LIN {X 0,Y 297.727,Z 299.631,A -85,B 0,C 180,E1 -16461.174,E2 -16461.174} C_VEL
LIN {X 0,Y 297.211,Z 303.349,A -85,B 0,C 180,E1 -16463.293,E2 -16463.293} C_VEL
LIN {X 0,Y 297,Z 305.074,A -85,B 0,C 180,E1 -16464.569,E2 -16464.569} C_VEL
LIN {X 0,Y 296.826,Z 306.468,A -85,B 0,C 180,E1 -16465.927,E2 -16465.927} C_VEL
LIN {X 0,Y 296.548,Z 308.073,A -85,B 0,C 180,E1 -16468.642,E2 -16468.642} C_VEL
LIN {X 0,Y 296.529,Z 308.304,A -85,B 0,C 180,E1 -16470,E2 -16470} C_VEL
LIN {X 0,Y 296.548,Z 308.111,A -85,B 0,C 180,E1 -16471.358,E2 -16471.358} C_VEL
LIN {X 0,Y 296.821,Z 306.556,A -85,B 0,C 180,E1 -16474.074,E2 -16474.074} C_VEL
LIN {X 0,Y 296.965,Z 305.201,A -85,B 0,C 180,E1 -16475.432,E2 -16475.432} C_VEL
LIN {X 0,Y 297.36,Z 302.335,A -85,B 0,C 180,E1 -16477.469,E2 -16477.469} C_VEL
LIN {X 0,Y 297.904,Z 298.45,A -85,B 0,C 180,E1 -16479.506,E2 -16479.506} C_VEL
LIN {X 0,Y 298.767,Z 293.434,A -85,B 0,C 180,E1 -16481.534,E2 -16481.534} C_VEL
LIN {X 0,Y 299.934,Z 287.114,A -85,B 0,C 180,E1 -16483.552,E2 -16483.552} C_VEL
LIN {X 0,Y 301.351,Z 279.205,A -85,B 0,C 180,E1 -16485.557,E2 -16485.557} C_VEL
LIN {X 0,Y 302.82,Z 271.138,A -85,B 0,C 180,E1 -16487.212,E2 -16487.212} C_VEL
LIN {X 0,Y 304.186,Z 261.302,A -85,B 0,C 180,E1 -16488.873,E2 -16488.873} C_VEL
LIN {X 0,Y 305.736,Z 250.222,A -85,B 0,C 180,E1 -16490.346,E2 -16490.346} C_VEL
LIN {X 0,Y 306.69,Z 242.741,A -85,B 0,C 180,E1 -16491.157,E2 -16491.157} C_VEL
LIN {X 0,Y 305.142,Z 232.366,A -85,B 0,C 180,E1 -16492.291,E2 -16492.291} C_VEL
LIN {X 0,Y 302.504,Z 220.449,A -85,B 0,C 180,E1 -16493.406,E2 -16493.406} C_VEL
LIN {X 0,Y 298.984,Z 208.375,A -85,B 0,C 180,E1 -16494.349,E2 -16494.349} C_VEL
LIN {X 0,Y 297.712,Z 203.982,A -85,B 0,C 180,E1 -16494.644,E2 -16494.644} C_VEL
LIN {X 0,Y 297.998,Z 200.351,A -85,B 0,C 180,E1 -16498.144,E2 -16498.144} C_VEL
LIN {X 0,Y 298.334,Z 196.579,A -85,B 0,C 180,E1 -16501.997,E2 -16501.997} C_VEL
LIN {X 0,Y 298.503,Z 194.178,A -85,B 0,C 180,E1 -16504.508,E2 -16504.508} C_VEL
LIN {X 0,Y 298.467,Z 191.246,A -85,B 0,C 180,E1 -16507.751,E2 -16507.751} C_VEL
LIN {X 0,Y 298.356,Z 190.321,A -85,B 0,C 180,E1 -16508.982,E2 -16508.982} C_VEL
LIN {X 0,Y 298.372,Z 190.319,A -85,B 0,C 180,E1 -16513.097,E2 -16513.097} C_VEL
LIN {X 0,Y 298.404,Z 190.316,A -85,B 0,C 180,E1 -16516.921,E2 -16516.921} C_VEL
LIN {X 0,Y 298.397,Z 190.317,A -85,B 0,C 180,E1 -16521.008,E2 -16521.008} C_VEL
LIN {X 0,Y 298.406,Z 190.313,A -85,B 0,C 180,E1 -16523.928,E2 -16523.928} C_VEL
LIN {X 0,Y 298.396,Z 190.313,A -85,B 0,C 180,E1 -16527.2,E2 -16527.2} C_VEL
LIN {X 0,Y 298.428,Z 190.312,A -85,B 0,C 180,E1 -16530.616,E2 -16530.616} C_VEL
LIN {X 0,Y 298.48,Z 190.302,A -85,B 0,C 180,E1 -16533.476,E2 -16533.476} C_VEL
LIN {X 0,Y 298.437,Z 190.309,A -85,B 0,C 180,E1 -16536.697,E2 -16536.697} C_VEL
LIN {X 0,Y 298.541,Z 190.295,A -85,B 0,C 180,E1 -16540.757,E2 -16540.757} C_VEL
LIN {X 0,Y 298.595,Z 190.289,A -85,B 0,C 180,E1 -16544.995,E2 -16544.995} C_VEL
LIN {X 0,Y 298.584,Z 190.291,A -85,B 0,C 180,E1 -16549.146,E2 -16549.146} C_VEL
LIN {X 0,Y 298.706,Z 190.276,A -85,B 0,C 180,E1 -16551.229,E2 -16551.229} C_VEL
LIN {X 0,Y 297.983,Z 190.365,A -85,B 0,C 180,E1 -16552.353,E2 -16552.353} C_VEL
LIN {X 0,Y 295.038,Z 190.732,A -85,B 0,C 180,E1 -16554.182,E2 -16554.182} C_VEL
LIN {X 0,Y 292.659,Z 191.031,A -85,B 0,C 180,E1 -16555.668,E2 -16555.668} C_VEL
LIN {X 0,Y 291.776,Z 191.14,A -85,B 0,C 180,E1 -16556.819,E2 -16556.819} C_VEL
LIN {X 0,Y 291.777,Z 191.142,A -85,B 0,C 180,E1 -16557.208,E2 -16557.208} C_VEL
LIN {X 0,Y 291.968,Z 191.114,A -85,B 0,C 180,E1 -16560,E2 -16560} C_VEL
LIN {X 0,Y 291.786,Z 191.139,A -85,B 0,C 180,E1 -16562.761,E2 -16562.761} C_VEL
LIN {X 0,Y 291.688,Z 191.154,A -85,B 0,C 180,E1 -16566.919,E2 -16566.919} C_VEL
LIN {X 0,Y 291.574,Z 191.164,A -85,B 0,C 180,E1 -16569.714,E2 -16569.714} C_VEL
LIN {X 0,Y 291.524,Z 191.171,A -85,B 0,C 180,E1 -16573.95,E2 -16573.95} C_VEL
LIN {X 0,Y 291.488,Z 191.177,A -85,B 0,C 180,E1 -16576.818,E2 -16576.818} C_VEL
LIN {X 0,Y 291.452,Z 191.181,A -85,B 0,C 180,E1 -16579.875,E2 -16579.875} C_VEL
LIN {X 0,Y 291.384,Z 191.191,A -85,B 0,C 180,E1 -16584.207,E2 -16584.207} C_VEL
LIN {X 0,Y 291.422,Z 191.183,A -85,B 0,C 180,E1 -16587.272,E2 -16587.272} C_VEL
LIN {X 0,Y 291.335,Z 191.196,A -85,B 0,C 180,E1 -16590.437,E2 -16590.437} C_VEL
LIN {X 0,Y 291.345,Z 191.197,A -85,B 0,C 180,E1 -16593.698,E2 -16593.698} C_VEL
LIN {X 0,Y 291.36,Z 191.194,A -85,B 0,C 180,E1 -16597.25,E2 -16597.25} C_VEL
LIN {X 0,Y 291.333,Z 191.197,A -85,B 0,C 180,E1 -16600.643,E2 -16600.643} C_VEL
LIN {X 0,Y 291.398,Z 191.4,A -85,B 0,C 180,E1 -16602.478,E2 -16602.478} C_VEL
LIN {X 0,Y 292.043,Z 195.349,A -85,B 0,C 180,E1 -16606.216,E2 -16606.216} C_VEL
LIN {X 0,Y 292.729,Z 199.137,A -85,B 0,C 180,E1 -16609.591,E2 -16609.591} C_VEL
LIN {X 0,Y 293.088,Z 202.423,A -85,B 0,C 180,E1 -16612.309,E2 -16612.309} C_VEL
LIN {X 0,Y 293.108,Z 205.65,A -85,B 0,C 180,E1 -16614.868,E2 -16614.868} C_VEL
LIN {X 0,Y 292.471,Z 209.913,A -85,B 0,C 180,E1 -16618.085,E2 -16618.085} C_VEL
LIN {X 0,Y 291.733,Z 215.231,A -85,B 0,C 180,E1 -16621.981,E2 -16621.981} C_VEL
LIN {X 0,Y 291.179,Z 219.113,A -85,B 0,C 180,E1 -16624.786,E2 -16624.786} C_VEL
LIN {X 0,Y 294.511,Z 233.044,A -85,B 0,C 180,E1 -16625.735,E2 -16625.735} C_VEL
LIN {X 0,Y 296.711,Z 245.302,A -85,B 0,C 180,E1 -16626.774,E2 -16626.774} C_VEL
LIN {X 0,Y 298.14,Z 257.517,A -85,B 0,C 180,E1 -16628.024,E2 -16628.024} C_VEL
LIN {X 0,Y 298.59,Z 265.376,A -85,B 0,C 180,E1 -16628.964,E2 -16628.964} C_VEL
LIN {X 0,Y 296.793,Z 276.914,A -85,B 0,C 180,E1 -16630.459,E2 -16630.459} C_VEL
LIN {X 0,Y 295.278,Z 286.212,A -85,B 0,C 180,E1 -16631.976,E2 -16631.976} C_VEL
LIN {X 0,Y 293.884,Z 294.693,A -85,B 0,C 180,E1 -16633.68,E2 -16633.68} C_VEL
LIN {X 0,Y 292.416,Z 302.971,A -85,B 0,C 180,E1 -16635.738,E2 -16635.738} C_VEL
LIN {X 0,Y 291.205,Z 309.644,A -85,B 0,C 180,E1 -16637.809,E2 -16637.809} C_VEL
LIN {X 0,Y 290.315,Z 315.757,A -85,B 0,C 180,E1 -16640.243,E2 -16640.243} C_VEL
LIN {X 0,Y 289.813,Z 319.731,A -85,B 0,C 180,E1 -16642.335,E2 -16642.335} C_VEL
LIN {X 0,Y 289.517,Z 322.668,A -85,B 0,C 180,E1 -16644.428,E2 -16644.428} C_VEL
LIN {X 0,Y 289.45,Z 324.067,A -85,B 0,C 180,E1 -16645.822,E2 -16645.822} C_VEL
LIN {X 0,Y 289.441,Z 325.067,A -85,B 0,C 180,E1 -16647.216,E2 -16647.216} C_VEL
LIN {X 0,Y 289.403,Z 325.676,A -85,B 0,C 180,E1 -16648.608,E2 -16648.608} C_VEL
LIN {X 0,Y 289.406,Z 325.891,A -85,B 0,C 180,E1 -16650,E2 -16650} C_VEL
LIN {X 0,Y 289.403,Z 325.671,A -85,B 0,C 180,E1 -16651.391,E2 -16651.391} C_VEL
LIN {X 0,Y 289.441,Z 325.061,A -85,B 0,C 180,E1 -16652.783,E2 -16652.783} C_VEL
LIN {X 0,Y 289.45,Z 324.059,A -85,B 0,C 180,E1 -16654.177,E2 -16654.177} C_VEL
LIN {X 0,Y 289.517,Z 322.655,A -85,B 0,C 180,E1 -16655.572,E2 -16655.572} C_VEL
LIN {X 0,Y 289.812,Z 319.709,A -85,B 0,C 180,E1 -16657.664,E2 -16657.664} C_VEL
LIN {X 0,Y 290.315,Z 315.724,A -85,B 0,C 180,E1 -16659.756,E2 -16659.756} C_VEL
LIN {X 0,Y 291.204,Z 309.6,A -85,B 0,C 180,E1 -16662.191,E2 -16662.191} C_VEL
LIN {X 0,Y 292.411,Z 302.916,A -85,B 0,C 180,E1 -16664.262,E2 -16664.262} C_VEL
LIN {X 0,Y 293.887,Z 294.626,A -85,B 0,C 180,E1 -16666.319,E2 -16666.319} C_VEL
LIN {X 0,Y 295.283,Z 286.126,A -85,B 0,C 180,E1 -16668.023,E2 -16668.023} C_VEL
LIN {X 0,Y 296.957,Z 275.627,A -85,B 0,C 180,E1 -16669.709,E2 -16669.709} C_VEL
LIN {X 0,Y 298.51,Z 265.243,A -85,B 0,C 180,E1 -16671.041,E2 -16671.041} C_VEL
LIN {X 0,Y 297.778,Z 253.852,A -85,B 0,C 180,E1 -16672.362,E2 -16672.362} C_VEL
LIN {X 0,Y 296.103,Z 241.278,A -85,B 0,C 180,E1 -16673.568,E2 -16673.568} C_VEL
LIN {X 0,Y 293.608,Z 228.856,A -85,B 0,C 180,E1 -16674.55,E2 -16674.55} C_VEL
LIN {X 0,Y 291.202,Z 219.121,A -85,B 0,C 180,E1 -16675.186,E2 -16675.186} C_VEL
LIN {X 0,Y 291.862,Z 214.156,A -85,B 0,C 180,E1 -16678.789,E2 -16678.789} C_VEL
LIN {X 0,Y 292.469,Z 209.901,A -85,B 0,C 180,E1 -16681.914,E2 -16681.914} C_VEL
LIN {X 0,Y 293.131,Z 205.279,A -85,B 0,C 180,E1 -16685.395,E2 -16685.395} C_VEL
LIN {X 0,Y 293.067,Z 201.302,A -85,B 0,C 180,E1 -16688.572,E2 -16688.572} C_VEL
LIN {X 0,Y 292.361,Z 196.965,A -85,B 0,C 180,E1 -16692.305,E2 -16692.305} C_VEL
LIN {X 0,Y 291.589,Z 192.61,A -85,B 0,C 180,E1 -16696.308,E2 -16696.308} C_VEL
LIN {X 0,Y 291.361,Z 191.198,A -85,B 0,C 180,E1 -16697.767,E2 -16697.767} C_VEL
LIN {X 0,Y 291.342,Z 191.195,A -85,B 0,C 180,E1 -16701.156,E2 -16701.156} C_VEL
LIN {X 0,Y 291.353,Z 191.195,A -85,B 0,C 180,E1 -16704.625,E2 -16704.625} C_VEL
LIN {X 0,Y 291.369,Z 191.193,A -85,B 0,C 180,E1 -16707.95,E2 -16707.95} C_VEL
LIN {X 0,Y 291.375,Z 191.188,A -85,B 0,C 180,E1 -16711.158,E2 -16711.158} C_VEL
LIN {X 0,Y 291.413,Z 191.187,A -85,B 0,C 180,E1 -16714.272,E2 -16714.272} C_VEL
LIN {X 0,Y 291.372,Z 191.191,A -85,B 0,C 180,E1 -16717.299,E2 -16717.299} C_VEL
LIN {X 0,Y 291.456,Z 191.18,A -85,B 0,C 180,E1 -16720.27,E2 -16720.27} C_VEL
LIN {X 0,Y 291.553,Z 191.166,A -85,B 0,C 180,E1 -16724.624,E2 -16724.624} C_VEL
LIN {X 0,Y 291.527,Z 191.17,A -85,B 0,C 180,E1 -16728.88,E2 -16728.88} C_VEL
LIN {X 0,Y 291.649,Z 191.155,A -85,B 0,C 180,E1 -16731.687,E2 -16731.687} C_VEL
LIN {X 0,Y 291.604,Z 191.16,A -85,B 0,C 180,E1 -16734.468,E2 -16734.468} C_VEL
LIN {X 0,Y 291.887,Z 191.126,A -85,B 0,C 180,E1 -16738.62,E2 -16738.62} C_VEL
LIN {X 0,Y 291.887,Z 191.125,A -85,B 0,C 180,E1 -16741.38,E2 -16741.38} C_VEL
LIN {X 0,Y 291.652,Z 191.153,A -85,B 0,C 180,E1 -16746.606,E2 -16746.606} C_VEL
LIN {X 0,Y 291.566,Z 191.164,A -85,B 0,C 180,E1 -16749.714,E2 -16749.714} C_VEL
LIN {X 0,Y 291.52,Z 191.172,A -85,B 0,C 180,E1 -16753.95,E2 -16753.95} C_VEL
LIN {X 0,Y 291.485,Z 191.175,A -85,B 0,C 180,E1 -16756.818,E2 -16756.818} C_VEL
LIN {X 0,Y 291.449,Z 191.182,A -85,B 0,C 180,E1 -16759.875,E2 -16759.875} C_VEL
LIN {X 0,Y 291.399,Z 191.187,A -85,B 0,C 180,E1 -16764.206,E2 -16764.206} C_VEL
LIN {X 0,Y 291.42,Z 191.184,A -85,B 0,C 180,E1 -16767.272,E2 -16767.272} C_VEL
LIN {X 0,Y 291.336,Z 191.193,A -85,B 0,C 180,E1 -16770.437,E2 -16770.437} C_VEL
LIN {X 0,Y 291.343,Z 191.195,A -85,B 0,C 180,E1 -16773.699,E2 -16773.699} C_VEL
LIN {X 0,Y 291.358,Z 191.193,A -85,B 0,C 180,E1 -16777.25,E2 -16777.25} C_VEL
LIN {X 0,Y 291.331,Z 191.196,A -85,B 0,C 180,E1 -16780.643,E2 -16780.643} C_VEL
LIN {X 0,Y 291.289,Z 191.201,A -85,B 0,C 180,E1 -16784.402,E2 -16784.402} C_VEL
LIN {X 0,Y 291.326,Z 191.198,A -85,B 0,C 180,E1 -16788.405,E2 -16788.405} C_VEL
LIN {X 0,Y 291.354,Z 191.329,A -85,B 0,C 180,E1 -16791.159,E2 -16791.159} C_VEL
LIN {X 0,Y 291.48,Z 192.836,A -85,B 0,C 180,E1 -16792.931,E2 -16792.931} C_VEL
LIN {X 0,Y 291.385,Z 195.862,A -85,B 0,C 180,E1 -16796.308,E2 -16796.308} C_VEL
LIN {X 0,Y 291.133,Z 198.907,A -85,B 0,C 180,E1 -16799.54,E2 -16799.54} C_VEL
LIN {X 0,Y 290.825,Z 202.734,A -85,B 0,C 180,E1 -16803.398,E2 -16803.398} C_VEL
LIN {X 0,Y 290.713,Z 204.19,A -85,B 0,C 180,E1 -16804.833,E2 -16804.833} C_VEL
LIN {X 0,Y 295.103,Z 218.824,A -85,B 0,C 180,E1 -16805.974,E2 -16805.974} C_VEL
LIN {X 0,Y 297.738,Z 229.936,A -85,B 0,C 180,E1 -16807.012,E2 -16807.012} C_VEL
LIN {X 0,Y 299.765,Z 241.957,A -85,B 0,C 180,E1 -16808.331,E2 -16808.331} C_VEL
LIN {X 0,Y 299.595,Z 246.67,A -85,B 0,C 180,E1 -16808.859,E2 -16808.859} C_VEL
LIN {X 0,Y 298.065,Z 257.33,A -85,B 0,C 180,E1 -16810.188,E2 -16810.188} C_VEL
LIN {X 0,Y 296.646,Z 267.314,A -85,B 0,C 180,E1 -16811.757,E2 -16811.757} C_VEL
LIN {X 0,Y 295.145,Z 275.868,A -85,B 0,C 180,E1 -16813.397,E2 -16813.397} C_VEL
LIN {X 0,Y 293.51,Z 284.483,A -85,B 0,C 180,E1 -16815.439,E2 -16815.439} C_VEL
LIN {X 0,Y 292.236,Z 291.349,A -85,B 0,C 180,E1 -16817.5,E2 -16817.5} C_VEL
LIN {X 0,Y 291.199,Z 296.845,A -85,B 0,C 180,E1 -16819.572,E2 -16819.572} C_VEL
LIN {X 0,Y 290.493,Z 301.155,A -85,B 0,C 180,E1 -16821.654,E2 -16821.654} C_VEL
LIN {X 0,Y 290.13,Z 303.823,A -85,B 0,C 180,E1 -16823.301,E2 -16823.301} C_VEL
LIN {X 0,Y 289.747,Z 306.682,A -85,B 0,C 180,E1 -16825.827,E2 -16825.827} C_VEL
LIN {X 0,Y 289.469,Z 308.286,A -85,B 0,C 180,E1 -16828.609,E2 -16828.609} C_VEL
LIN {X 0,Y 289.447,Z 308.516,A -85,B 0,C 180,E1 -16830,E2 -16830} C_VEL
LIN {X 0,Y 289.469,Z 308.324,A -85,B 0,C 180,E1 -16831.392,E2 -16831.392} C_VEL
LIN {X 0,Y 289.74,Z 306.769,A -85,B 0,C 180,E1 -16834.173,E2 -16834.173} C_VEL
LIN {X 0,Y 290.12,Z 304.006,A -85,B 0,C 180,E1 -16836.682,E2 -16836.682} C_VEL
LIN {X 0,Y 290.668,Z 300.075,A -85,B 0,C 180,E1 -16839.043,E2 -16839.043} C_VEL
LIN {X 0,Y 291.48,Z 295.443,A -85,B 0,C 180,E1 -16841.122,E2 -16841.122} C_VEL
LIN {X 0,Y 292.84,Z 288.456,A -85,B 0,C 180,E1 -16843.533,E2 -16843.533} C_VEL
LIN {X 0,Y 294.227,Z 280.885,A -85,B 0,C 180,E1 -16845.588,E2 -16845.588} C_VEL
LIN {X 0,Y 295.73,Z 273.121,A -85,B 0,C 180,E1 -16847.281,E2 -16847.281} C_VEL
LIN {X 0,Y 297.252,Z 263.03,A -85,B 0,C 180,E1 -16849.074,E2 -16849.074} C_VEL
LIN {X 0,Y 298.885,Z 251.822,A -85,B 0,C 180,E1 -16850.653,E2 -16850.653} C_VEL
LIN {X 0,Y 299.937,Z 244.524,A -85,B 0,C 180,E1 -16851.477,E2 -16851.477} C_VEL
LIN {X 0,Y 298.636,Z 234.606,A -85,B 0,C 180,E1 -16852.616,E2 -16852.616} C_VEL
LIN {X 0,Y 296.103,Z 222.751,A -85,B 0,C 180,E1 -16853.797,E2 -16853.797} C_VEL
LIN {X 0,Y 292.7,Z 210.604,A -85,B 0,C 180,E1 -16854.818,E2 -16854.818} C_VEL
LIN {X 0,Y 290.721,Z 204.203,A -85,B 0,C 180,E1 -16855.275,E2 -16855.275} C_VEL
LIN {X 0,Y 291.121,Z 199.817,A -85,B 0,C 180,E1 -16859.647,E2 -16859.647} C_VEL
LIN {X 0,Y 291.32,Z 197.203,A -85,B 0,C 180,E1 -16862.396,E2 -16862.396} C_VEL
LIN {X 0,Y 291.494,Z 194.483,A -85,B 0,C 180,E1 -16865.356,E2 -16865.356} C_VEL
LIN {X 0,Y 291.494,Z 192.763,A -85,B 0,C 180,E1 -16867.284,E2 -16867.284} C_VEL
LIN {X 0,Y 291.314,Z 191.198,A -85,B 0,C 180,E1 -16869.465,E2 -16869.465} C_VEL
LIN {X 0,Y 291.291,Z 191.199,A -85,B 0,C 180,E1 -16873.629,E2 -16873.629} C_VEL
LIN {X 0,Y 291.321,Z 191.196,A -85,B 0,C 180,E1 -16877.508,E2 -16877.508} C_VEL
LIN {X 0,Y 291.345,Z 191.195,A -85,B 0,C 180,E1 -16881.157,E2 -16881.157} C_VEL
LIN {X 0,Y 291.356,Z 191.194,A -85,B 0,C 180,E1 -16884.625,E2 -16884.625} C_VEL
LIN {X 0,Y 291.372,Z 191.188,A -85,B 0,C 180,E1 -16887.951,E2 -16887.951} C_VEL
LIN {X 0,Y 291.379,Z 191.188,A -85,B 0,C 180,E1 -16891.158,E2 -16891.158} C_VEL
LIN {X 0,Y 291.416,Z 191.185,A -85,B 0,C 180,E1 -16894.272,E2 -16894.272} C_VEL
LIN {X 0,Y 291.383,Z 191.186,A -85,B 0,C 180,E1 -16897.3,E2 -16897.3} C_VEL
LIN {X 0,Y 291.459,Z 191.18,A -85,B 0,C 180,E1 -16900.27,E2 -16900.27} C_VEL
LIN {X 0,Y 291.557,Z 191.166,A -85,B 0,C 180,E1 -16904.624,E2 -16904.624} C_VEL
LIN {X 0,Y 291.53,Z 191.169,A -85,B 0,C 180,E1 -16908.88,E2 -16908.88} C_VEL
LIN {X 0,Y 291.653,Z 191.157,A -85,B 0,C 180,E1 -16911.687,E2 -16911.687} C_VEL
LIN {X 0,Y 291.606,Z 191.159,A -85,B 0,C 180,E1 -16914.468,E2 -16914.468} C_VEL
LIN {X 0,Y 291.777,Z 191.142,A -85,B 0,C 180,E1 -16917.208,E2 -16917.208} C_VEL
LIN {X 0,Y 291.316,Z 191.207,A -85,B 0,C 180,E1 -16918.361,E2 -16918.361} C_VEL
LIN {X 0,Y 289.824,Z 191.395,A -85,B 0,C 180,E1 -16919.493,E2 -16919.493} C_VEL
LIN {X 0,Y 285.997,Z 191.865,A -85,B 0,C 180,E1 -16921.763,E2 -16921.763} C_VEL
LIN {X 0,Y 284.785,Z 192.012,A -85,B 0,C 180,E1 -16922.945,E2 -16922.945} C_VEL
LIN {X 0,Y 284.631,Z 192.028,A -85,B 0,C 180,E1 -16923.347,E2 -16923.347} C_VEL
LIN {X 0,Y 284.644,Z 192.03,A -85,B 0,C 180,E1 -16927.091,E2 -16927.091} C_VEL
LIN {X 0,Y 284.519,Z 192.043,A -85,B 0,C 180,E1 -16929.957,E2 -16929.957} C_VEL
LIN {X 0,Y 284.484,Z 192.05,A -85,B 0,C 180,E1 -16934.303,E2 -16934.303} C_VEL
LIN {X 0,Y 284.424,Z 192.055,A -85,B 0,C 180,E1 -16937.248,E2 -16937.248} C_VEL
LIN {X 0,Y 284.378,Z 192.064,A -85,B 0,C 180,E1 -16940.242,E2 -16940.242} C_VEL
LIN {X 0,Y 284.34,Z 192.066,A -85,B 0,C 180,E1 -16944.846,E2 -16944.846} C_VEL
LIN {X 0,Y 284.33,Z 192.07,A -85,B 0,C 180,E1 -16948.011,E2 -16948.011} C_VEL
LIN {X 0,Y 284.295,Z 192.073,A -85,B 0,C 180,E1 -16951.274,E2 -16951.274} C_VEL
LIN {X 0,Y 284.337,Z 192.069,A -85,B 0,C 180,E1 -16955.347,E2 -16955.347} C_VEL
LIN {X 0,Y 284.303,Z 192.072,A -85,B 0,C 180,E1 -16958.17,E2 -16958.17} C_VEL
LIN {X 0,Y 284.324,Z 192.194,A -85,B 0,C 180,E1 -16961.866,E2 -16961.866} C_VEL
LIN {X 0,Y 284.953,Z 196.04,A -85,B 0,C 180,E1 -16965.664,E2 -16965.664} C_VEL
LIN {X 0,Y 285.512,Z 198.966,A -85,B 0,C 180,E1 -16968.347,E2 -16968.347} C_VEL
LIN {X 0,Y 286.051,Z 202.974,A -85,B 0,C 180,E1 -16971.833,E2 -16971.833} C_VEL
LIN {X 0,Y 286.081,Z 205.811,A -85,B 0,C 180,E1 -16974.164,E2 -16974.164} C_VEL
LIN {X 0,Y 285.72,Z 209.108,A -85,B 0,C 180,E1 -16976.753,E2 -16976.753} C_VEL
LIN {X 0,Y 284.947,Z 213.976,A -85,B 0,C 180,E1 -16980.443,E2 -16980.443} C_VEL
LIN {X 0,Y 284.225,Z 218.888,A -85,B 0,C 180,E1 -16984.125,E2 -16984.125} C_VEL
LIN {X 0,Y 287.574,Z 232.389,A -85,B 0,C 180,E1 -16985.083,E2 -16985.083} C_VEL
LIN {X 0,Y 289.895,Z 245.209,A -85,B 0,C 180,E1 -16986.205,E2 -16986.205} C_VEL
LIN {X 0,Y 291.277,Z 257.3,A -85,B 0,C 180,E1 -16987.478,E2 -16987.478} C_VEL
LIN {X 0,Y 291.778,Z 266.597,A -85,B 0,C 180,E1 -16988.634,E2 -16988.634} C_VEL
LIN {X 0,Y 289.89,Z 277.835,A -85,B 0,C 180,E1 -16990.159,E2 -16990.159} C_VEL
LIN {X 0,Y 288.225,Z 287.619,A -85,B 0,C 180,E1 -16991.85,E2 -16991.85} C_VEL
LIN {X 0,Y 286.756,Z 295.973,A -85,B 0,C 180,E1 -16993.629,E2 -16993.629} C_VEL
LIN {X 0,Y 285.272,Z 303.996,A -85,B 0,C 180,E1 -16995.737,E2 -16995.737} C_VEL
LIN {X 0,Y 284.091,Z 310.429,A -85,B 0,C 180,E1 -16997.861,E2 -16997.861} C_VEL
LIN {X 0,Y 283.277,Z 315.543,A -85,B 0,C 180,E1 -16999.999,E2 -16999.999} C_VEL
LIN {X 0,Y 282.748,Z 319.517,A -85,B 0,C 180,E1 -17002.142,E2 -17002.142} C_VEL
LIN {X 0,Y 282.411,Z 322.7,A -85,B 0,C 180,E1 -17004.522,E2 -17004.522} C_VEL
LIN {X 0,Y 282.349,Z 324.854,A -85,B 0,C 180,E1 -17007.146,E2 -17007.146} C_VEL
LIN {X 0,Y 282.327,Z 325.464,A -85,B 0,C 180,E1 -17008.573,E2 -17008.573} C_VEL
LIN {X 0,Y 282.327,Z 325.679,A -85,B 0,C 180,E1 -17010,E2 -17010} C_VEL
LIN {X 0,Y 282.327,Z 325.459,A -85,B 0,C 180,E1 -17011.426,E2 -17011.426} C_VEL
LIN {X 0,Y 282.349,Z 324.847,A -85,B 0,C 180,E1 -17012.853,E2 -17012.853} C_VEL
LIN {X 0,Y 282.41,Z 322.687,A -85,B 0,C 180,E1 -17015.477,E2 -17015.477} C_VEL
LIN {X 0,Y 282.747,Z 319.494,A -85,B 0,C 180,E1 -17017.857,E2 -17017.857} C_VEL
LIN {X 0,Y 283.277,Z 315.509,A -85,B 0,C 180,E1 -17020.001,E2 -17020.001} C_VEL
LIN {X 0,Y 284.229,Z 309.384,A -85,B 0,C 180,E1 -17022.495,E2 -17022.495} C_VEL
LIN {X 0,Y 285.505,Z 302.7,A -85,B 0,C 180,E1 -17024.614,E2 -17024.614} C_VEL
LIN {X 0,Y 287.07,Z 294.411,A -85,B 0,C 180,E1 -17026.718,E2 -17026.718} C_VEL
LIN {X 0,Y 288.502,Z 285.909,A -85,B 0,C 180,E1 -17028.462,E2 -17028.462} C_VEL
LIN {X 0,Y 290.274,Z 275.41,A -85,B 0,C 180,E1 -17030.182,E2 -17030.182} C_VEL
LIN {X 0,Y 291.699,Z 266.454,A -85,B 0,C 180,E1 -17031.371,E2 -17031.371} C_VEL
LIN {X 0,Y 291.107,Z 255.338,A -85,B 0,C 180,E1 -17032.723,E2 -17032.723} C_VEL
LIN {X 0,Y 289.484,Z 242.591,A -85,B 0,C 180,E1 -17034.026,E2 -17034.026} C_VEL
LIN {X 0,Y 287.059,Z 230.308,A -85,B 0,C 180,E1 -17035.06,E2 -17035.06} C_VEL
LIN {X 0,Y 284.235,Z 218.857,A -85,B 0,C 180,E1 -17035.875,E2 -17035.875} C_VEL
LIN {X 0,Y 284.945,Z 213.946,A -85,B 0,C 180,E1 -17039.556,E2 -17039.556} C_VEL
LIN {X 0,Y 285.718,Z 209.086,A -85,B 0,C 180,E1 -17043.246,E2 -17043.246} C_VEL
LIN {X 0,Y 286.086,Z 205.422,A -85,B 0,C 180,E1 -17046.127,E2 -17046.127} C_VEL
LIN {X 0,Y 286.076,Z 202.93,A -85,B 0,C 180,E1 -17048.173,E2 -17048.173} C_VEL
LIN {X 0,Y 285.51,Z 198.939,A -85,B 0,C 180,E1 -17051.653,E2 -17051.653} C_VEL
LIN {X 0,Y 284.742,Z 194.585,A -85,B 0,C 180,E1 -17055.706,E2 -17055.706} C_VEL
LIN {X 0,Y 284.31,Z 192.075,A -85,B 0,C 180,E1 -17058.368,E2 -17058.368} C_VEL
LIN {X 0,Y 284.309,Z 192.072,A -85,B 0,C 180,E1 -17062.281,E2 -17062.281} C_VEL
LIN {X 0,Y 284.305,Z 192.07,A -85,B 0,C 180,E1 -17065.35,E2 -17065.35} C_VEL
LIN {X 0,Y 284.292,Z 192.072,A -85,B 0,C 180,E1 -17068.725,E2 -17068.725} C_VEL
LIN {X 0,Y 284.394,Z 192.059,A -85,B 0,C 180,E1 -17072.827,E2 -17072.827} C_VEL
LIN {X 0,Y 284.331,Z 192.067,A -85,B 0,C 180,E1 -17076.704,E2 -17076.704} C_VEL
LIN {X 0,Y 284.402,Z 192.06,A -85,B 0,C 180,E1 -17081.261,E2 -17081.261} C_VEL
LIN {X 0,Y 284.49,Z 192.046,A -85,B 0,C 180,E1 -17084.459,E2 -17084.459} C_VEL
LIN {X 0,Y 284.48,Z 192.046,A -85,B 0,C 180,E1 -17088.601,E2 -17088.601} C_VEL
LIN {X 0,Y 284.606,Z 192.034,A -85,B 0,C 180,E1 -17091.48,E2 -17091.48} C_VEL
LIN {X 0,Y 284.573,Z 192.036,A -85,B 0,C 180,E1 -17094.331,E2 -17094.331} C_VEL
LIN {X 0,Y 284.853,Z 192.002,A -85,B 0,C 180,E1 -17098.586,E2 -17098.586} C_VEL
LIN {X 0,Y 284.853,Z 192.001,A -85,B 0,C 180,E1 -17101.414,E2 -17101.414} C_VEL
LIN {X 0,Y 284.64,Z 192.028,A -85,B 0,C 180,E1 -17107.092,E2 -17107.092} C_VEL
LIN {X 0,Y 284.512,Z 192.044,A -85,B 0,C 180,E1 -17109.957,E2 -17109.957} C_VEL
LIN {X 0,Y 284.48,Z 192.051,A -85,B 0,C 180,E1 -17114.303,E2 -17114.303} C_VEL
LIN {X 0,Y 284.424,Z 192.054,A -85,B 0,C 180,E1 -17117.249,E2 -17117.249} C_VEL
LIN {X 0,Y 284.377,Z 192.062,A -85,B 0,C 180,E1 -17120.242,E2 -17120.242} C_VEL
LIN {X 0,Y 284.368,Z 192.065,A -85,B 0,C 180,E1 -17123.876,E2 -17123.876} C_VEL
LIN {X 0,Y 284.394,Z 192.059,A -85,B 0,C 180,E1 -17127.173,E2 -17127.173} C_VEL
LIN {X 0,Y 284.295,Z 192.073,A -85,B 0,C 180,E1 -17131.275,E2 -17131.275} C_VEL
LIN {X 0,Y 284.335,Z 192.069,A -85,B 0,C 180,E1 -17135.347,E2 -17135.347} C_VEL
LIN {X 0,Y 284.301,Z 192.071,A -85,B 0,C 180,E1 -17138.171,E2 -17138.171} C_VEL
LIN {X 0,Y 284.268,Z 192.074,A -85,B 0,C 180,E1 -17142.125,E2 -17142.125} C_VEL
LIN {X 0,Y 284.254,Z 192.076,A -85,B 0,C 180,E1 -17146.19,E2 -17146.19} C_VEL
LIN {X 0,Y 284.306,Z 192.072,A -85,B 0,C 180,E1 -17150.025,E2 -17150.025} C_VEL
LIN {X 0,Y 284.427,Z 193.375,A -85,B 0,C 180,E1 -17152.251,E2 -17152.251} C_VEL
LIN {X 0,Y 284.404,Z 196.064,A -85,B 0,C 180,E1 -17155.365,E2 -17155.365} C_VEL
LIN {X 0,Y 284.164,Z 199.123,A -85,B 0,C 180,E1 -17158.71,E2 -17158.71} C_VEL
LIN {X 0,Y 283.886,Z 202.211,A -85,B 0,C 180,E1 -17161.942,E2 -17161.942} C_VEL
LIN {X 0,Y 283.737,Z 204.425,A -85,B 0,C 180,E1 -17164.182,E2 -17164.182} C_VEL
LIN {X 0,Y 285.955,Z 211.559,A -85,B 0,C 180,E1 -17164.716,E2 -17164.716} C_VEL
LIN {X 0,Y 289.185,Z 222.637,A -85,B 0,C 180,E1 -17165.692,E2 -17165.692} C_VEL
LIN {X 0,Y 291.712,Z 234.64,A -85,B 0,C 180,E1 -17166.918,E2 -17166.918} C_VEL
LIN {X 0,Y 293.132,Z 243.754,A -85,B 0,C 180,E1 -17168,E2 -17168} C_VEL
LIN {X 0,Y 292.577,Z 249.746,A -85,B 0,C 180,E1 -17168.696,E2 -17168.696} C_VEL
LIN {X 0,Y 290.842,Z 261.042,A -85,B 0,C 180,E1 -17170.227,E2 -17170.227} C_VEL
LIN {X 0,Y 289.34,Z 270.998,A -85,B 0,C 180,E1 -17171.96,E2 -17171.96} C_VEL
LIN {X 0,Y 287.461,Z 280.636,A -85,B 0,C 180,E1 -17174.036,E2 -17174.036} C_VEL
LIN {X 0,Y 285.973,Z 288.317,A -85,B 0,C 180,E1 -17176.137,E2 -17176.137} C_VEL
LIN {X 0,Y 284.555,Z 295.368,A -85,B 0,C 180,E1 -17178.605,E2 -17178.605} C_VEL
LIN {X 0,Y 283.681,Z 300.06,A -85,B 0,C 180,E1 -17180.734,E2 -17180.734} C_VEL
LIN {X 0,Y 283.042,Z 304.293,A -85,B 0,C 180,E1 -17183.322,E2 -17183.322} C_VEL
LIN {X 0,Y 282.67,Z 306.895,A -85,B 0,C 180,E1 -17185.723,E2 -17185.723} C_VEL
LIN {X 0,Y 282.392,Z 308.499,A -85,B 0,C 180,E1 -17188.574,E2 -17188.574} C_VEL
LIN {X 0,Y 282.367,Z 308.729,A -85,B 0,C 180,E1 -17190,E2 -17190} C_VEL
LIN {X 0,Y 282.392,Z 308.536,A -85,B 0,C 180,E1 -17191.426,E2 -17191.426} C_VEL
LIN {X 0,Y 282.662,Z 306.981,A -85,B 0,C 180,E1 -17194.278,E2 -17194.278} C_VEL
LIN {X 0,Y 283.018,Z 304.485,A -85,B 0,C 180,E1 -17196.637,E2 -17196.637} C_VEL
LIN {X 0,Y 283.665,Z 300.287,A -85,B 0,C 180,E1 -17199.268,E2 -17199.268} C_VEL
LIN {X 0,Y 284.518,Z 295.655,A -85,B 0,C 180,E1 -17201.398,E2 -17201.398} C_VEL
LIN {X 0,Y 285.936,Z 288.668,A -85,B 0,C 180,E1 -17203.866,E2 -17203.866} C_VEL
LIN {X 0,Y 287.409,Z 281.095,A -85,B 0,C 180,E1 -17205.968,E2 -17205.968} C_VEL
LIN {X 0,Y 288.974,Z 273.33,A -85,B 0,C 180,E1 -17207.699,E2 -17207.699} C_VEL
LIN {X 0,Y 290.485,Z 263.562,A -85,B 0,C 180,E1 -17209.481,E2 -17209.481} C_VEL
LIN {X 0,Y 292.071,Z 253.319,A -85,B 0,C 180,E1 -17210.974,E2 -17210.974} C_VEL
LIN {X 0,Y 293.234,Z 244.735,A -85,B 0,C 180,E1 -17211.993,E2 -17211.993} C_VEL
LIN {X 0,Y 291.525,Z 233.511,A -85,B 0,C 180,E1 -17213.325,E2 -17213.325} C_VEL
LIN {X 0,Y 288.865,Z 221.417,A -85,B 0,C 180,E1 -17214.546,E2 -17214.546} C_VEL
LIN {X 0,Y 285.198,Z 209.323,A -85,B 0,C 180,E1 -17215.586,E2 -17215.586} C_VEL
LIN {X 0,Y 283.744,Z 204.402,A -85,B 0,C 180,E1 -17215.965,E2 -17215.965} C_VEL
LIN {X 0,Y 284.095,Z 200.432,A -85,B 0,C 180,E1 -17220.021,E2 -17220.021} C_VEL
LIN {X 0,Y 284.315,Z 197.729,A -85,B 0,C 180,E1 -17222.944,E2 -17222.944} C_VEL
LIN {X 0,Y 284.476,Z 195.541,A -85,B 0,C 180,E1 -17225.386,E2 -17225.386} C_VEL
LIN {X 0,Y 284.389,Z 193.155,A -85,B 0,C 180,E1 -17228.157,E2 -17228.157} C_VEL
LIN {X 0,Y 284.256,Z 192.076,A -85,B 0,C 180,E1 -17230.003,E2 -17230.003} C_VEL
LIN {X 0,Y 284.235,Z 192.077,A -85,B 0,C 180,E1 -17234.188,E2 -17234.188} C_VEL
LIN {X 0,Y 284.273,Z 192.073,A -85,B 0,C 180,E1 -17238.124,E2 -17238.124} C_VEL
LIN {X 0,Y 284.304,Z 192.07,A -85,B 0,C 180,E1 -17241.829,E2 -17241.829} C_VEL
LIN {X 0,Y 284.308,Z 192.069,A -85,B 0,C 180,E1 -17245.35,E2 -17245.35} C_VEL
LIN {X 0,Y 284.295,Z 192.073,A -85,B 0,C 180,E1 -17248.725,E2 -17248.725} C_VEL
LIN {X 0,Y 284.397,Z 192.058,A -85,B 0,C 180,E1 -17252.827,E2 -17252.827} C_VEL
LIN {X 0,Y 284.368,Z 192.061,A -85,B 0,C 180,E1 -17256.707,E2 -17256.707} C_VEL
LIN {X 0,Y 284.405,Z 192.056,A -85,B 0,C 180,E1 -17261.262,E2 -17261.262} C_VEL
LIN {X 0,Y 284.494,Z 192.046,A -85,B 0,C 180,E1 -17264.459,E2 -17264.459} C_VEL
LIN {X 0,Y 284.484,Z 192.046,A -85,B 0,C 180,E1 -17268.601,E2 -17268.601} C_VEL
LIN {X 0,Y 284.61,Z 192.034,A -85,B 0,C 180,E1 -17271.48,E2 -17271.48} C_VEL
LIN {X 0,Y 284.575,Z 192.035,A -85,B 0,C 180,E1 -17274.331,E2 -17274.331} C_VEL
LIN {X 0,Y 284.856,Z 192,A -85,B 0,C 180,E1 -17278.586,E2 -17278.586} C_VEL
LIN {X 0,Y 284.856,Z 192.003,A -85,B 0,C 180,E1 -17281.414,E2 -17281.414} C_VEL
LIN {X 0,Y 284.631,Z 192.028,A -85,B 0,C 180,E1 -17283.347,E2 -17283.347} C_VEL
LIN {X 0,Y 283.833,Z 192.13,A -85,B 0,C 180,E1 -17284.528,E2 -17284.528} C_VEL
LIN {X 0,Y 280.997,Z 192.483,A -85,B 0,C 180,E1 -17286.454,E2 -17286.454} C_VEL
LIN {X 0,Y 278.649,Z 192.776,A -85,B 0,C 180,E1 -17288.018,E2 -17288.018} C_VEL
LIN {X 0,Y 277.607,Z 192.906,A -85,B 0,C 180,E1 -17289.228,E2 -17289.228} C_VEL
LIN {X 0,Y 277.498,Z 192.917,A -85,B 0,C 180,E1 -17289.638,E2 -17289.638} C_VEL
LIN {X 0,Y 277.419,Z 192.929,A -85,B 0,C 180,E1 -17293.179,E2 -17293.179} C_VEL
LIN {X 0,Y 277.407,Z 192.932,A -85,B 0,C 180,E1 -17296.181,E2 -17296.181} C_VEL
LIN {X 0,Y 277.346,Z 192.939,A -85,B 0,C 180,E1 -17300.349,E2 -17300.349} C_VEL
LIN {X 0,Y 277.294,Z 192.946,A -85,B 0,C 180,E1 -17304.158,E2 -17304.158} C_VEL
LIN {X 0,Y 277.326,Z 192.941,A -85,B 0,C 180,E1 -17307.505,E2 -17307.505} C_VEL
LIN {X 0,Y 277.273,Z 192.948,A -85,B 0,C 180,E1 -17310.481,E2 -17310.481} C_VEL
LIN {X 0,Y 277.247,Z 192.954,A -85,B 0,C 180,E1 -17313.896,E2 -17313.896} C_VEL
LIN {X 0,Y 277.257,Z 192.951,A -85,B 0,C 180,E1 -17317.471,E2 -17317.471} C_VEL
LIN {X 0,Y 277.276,Z 192.979,A -85,B 0,C 180,E1 -17321.225,E2 -17321.225} C_VEL
LIN {X 0,Y 277.887,Z 196.775,A -85,B 0,C 180,E1 -17325.084,E2 -17325.084} C_VEL
LIN {X 0,Y 278.667,Z 201.09,A -85,B 0,C 180,E1 -17329.166,E2 -17329.166} C_VEL
LIN {X 0,Y 279.094,Z 205.253,A -85,B 0,C 180,E1 -17332.817,E2 -17332.817} C_VEL
LIN {X 0,Y 278.963,Z 208.454,A -85,B 0,C 180,E1 -17335.47,E2 -17335.47} C_VEL
LIN {X 0,Y 278.078,Z 213.765,A -85,B 0,C 180,E1 -17339.637,E2 -17339.637} C_VEL
LIN {X 0,Y 277.293,Z 218.688,A -85,B 0,C 180,E1 -17343.431,E2 -17343.431} C_VEL
LIN {X 0,Y 280.572,Z 231.761,A -85,B 0,C 180,E1 -17344.39,E2 -17344.39} C_VEL
LIN {X 0,Y 282.988,Z 244.506,A -85,B 0,C 180,E1 -17345.545,E2 -17345.545} C_VEL
LIN {X 0,Y 284.429,Z 256.688,A -85,B 0,C 180,E1 -17346.862,E2 -17346.862} C_VEL
LIN {X 0,Y 285.041,Z 266.417,A -85,B 0,C 180,E1 -17348.108,E2 -17348.108} C_VEL
LIN {X 0,Y 283.425,Z 276.495,A -85,B 0,C 180,E1 -17349.497,E2 -17349.497} C_VEL
LIN {X 0,Y 281.732,Z 285.789,A -85,B 0,C 180,E1 -17351.077,E2 -17351.077} C_VEL
LIN {X 0,Y 280.263,Z 294.271,A -85,B 0,C 180,E1 -17352.863,E2 -17352.863} C_VEL
LIN {X 0,Y 278.627,Z 302.547,A -85,B 0,C 180,E1 -17355.016,E2 -17355.016} C_VEL
LIN {X 0,Y 277.273,Z 309.219,A -85,B 0,C 180,E1 -17357.186,E2 -17357.186} C_VEL
LIN {X 0,Y 276.261,Z 315.33,A -85,B 0,C 180,E1 -17359.742,E2 -17359.742} C_VEL
LIN {X 0,Y 275.708,Z 319.305,A -85,B 0,C 180,E1 -17361.94,E2 -17361.94} C_VEL
LIN {X 0,Y 275.322,Z 322.691,A -85,B 0,C 180,E1 -17364.584,E2 -17364.584} C_VEL
LIN {X 0,Y 275.26,Z 324.642,A -85,B 0,C 180,E1 -17367.073,E2 -17367.073} C_VEL
LIN {X 0,Y 275.252,Z 325.251,A -85,B 0,C 180,E1 -17368.537,E2 -17368.537} C_VEL
LIN {X 0,Y 275.25,Z 325.466,A -85,B 0,C 180,E1 -17370,E2 -17370} C_VEL
LIN {X 0,Y 275.252,Z 325.246,A -85,B 0,C 180,E1 -17371.463,E2 -17371.463} C_VEL
LIN {X 0,Y 275.26,Z 324.634,A -85,B 0,C 180,E1 -17372.927,E2 -17372.927} C_VEL
LIN {X 0,Y 275.328,Z 322.663,A -85,B 0,C 180,E1 -17375.429,E2 -17375.429} C_VEL
LIN {X 0,Y 275.708,Z 319.28,A -85,B 0,C 180,E1 -17378.059,E2 -17378.059} C_VEL
LIN {X 0,Y 276.26,Z 315.294,A -85,B 0,C 180,E1 -17380.257,E2 -17380.257} C_VEL
LIN {X 0,Y 277.272,Z 309.168,A -85,B 0,C 180,E1 -17382.814,E2 -17382.814} C_VEL
LIN {X 0,Y 278.62,Z 302.485,A -85,B 0,C 180,E1 -17384.984,E2 -17384.984} C_VEL
LIN {X 0,Y 280.269,Z 294.195,A -85,B 0,C 180,E1 -17387.136,E2 -17387.136} C_VEL
LIN {X 0,Y 281.733,Z 285.692,A -85,B 0,C 180,E1 -17388.922,E2 -17388.922} C_VEL
LIN {X 0,Y 283.607,Z 275.193,A -85,B 0,C 180,E1 -17390.678,E2 -17390.678} C_VEL
LIN {X 0,Y 284.976,Z 266.283,A -85,B 0,C 180,E1 -17391.894,E2 -17391.894} C_VEL
LIN {X 0,Y 284.311,Z 255.11,A -85,B 0,C 180,E1 -17393.297,E2 -17393.297} C_VEL
LIN {X 0,Y 282.752,Z 242.864,A -85,B 0,C 180,E1 -17394.594,E2 -17394.594} C_VEL
LIN {X 0,Y 280.076,Z 229.561,A -85,B 0,C 180,E1 -17395.757,E2 -17395.757} C_VEL
LIN {X 0,Y 277.293,Z 218.654,A -85,B 0,C 180,E1 -17396.571,E2 -17396.571} C_VEL
LIN {X 0,Y 278.164,Z 213.184,A -85,B 0,C 180,E1 -17400.791,E2 -17400.791} C_VEL
LIN {X 0,Y 278.964,Z 208.435,A -85,B 0,C 180,E1 -17404.529,E2 -17404.529} C_VEL
LIN {X 0,Y 279.104,Z 205.217,A -85,B 0,C 180,E1 -17407.18,E2 -17407.18} C_VEL
LIN {X 0,Y 278.842,Z 202.064,A -85,B 0,C 180,E1 -17409.925,E2 -17409.925} C_VEL
LIN {X 0,Y 278.241,Z 198.717,A -85,B 0,C 180,E1 -17412.998,E2 -17412.998} C_VEL
LIN {X 0,Y 277.493,Z 194.399,A -85,B 0,C 180,E1 -17417.262,E2 -17417.262} C_VEL
LIN {X 0,Y 277.247,Z 192.953,A -85,B 0,C 180,E1 -17418.985,E2 -17418.985} C_VEL
LIN {X 0,Y 277.255,Z 192.951,A -85,B 0,C 180,E1 -17422.529,E2 -17422.529} C_VEL
LIN {X 0,Y 277.244,Z 192.952,A -85,B 0,C 180,E1 -17426.104,E2 -17426.104} C_VEL
LIN {X 0,Y 277.26,Z 192.948,A -85,B 0,C 180,E1 -17429.538,E2 -17429.538} C_VEL
LIN {X 0,Y 277.356,Z 192.936,A -85,B 0,C 180,E1 -17432.864,E2 -17432.864} C_VEL
LIN {X 0,Y 277.296,Z 192.946,A -85,B 0,C 180,E1 -17436.076,E2 -17436.076} C_VEL
LIN {X 0,Y 277.343,Z 192.937,A -85,B 0,C 180,E1 -17440.766,E2 -17440.766} C_VEL
LIN {X 0,Y 277.433,Z 192.929,A -85,B 0,C 180,E1 -17445.326,E2 -17445.326} C_VEL
LIN {X 0,Y 277.455,Z 192.922,A -85,B 0,C 180,E1 -17449.787,E2 -17449.787} C_VEL
LIN {X 0,Y 277.599,Z 192.906,A -85,B 0,C 180,E1 -17452.728,E2 -17452.728} C_VEL
LIN {X 0,Y 277.819,Z 192.878,A -85,B 0,C 180,E1 -17458.55,E2 -17458.55} C_VEL
LIN {X 0,Y 277.819,Z 192.877,A -85,B 0,C 180,E1 -17461.45,E2 -17461.45} C_VEL
LIN {X 0,Y 277.599,Z 192.904,A -85,B 0,C 180,E1 -17467.272,E2 -17467.272} C_VEL
LIN {X 0,Y 277.455,Z 192.924,A -85,B 0,C 180,E1 -17470.213,E2 -17470.213} C_VEL
LIN {X 0,Y 277.433,Z 192.926,A -85,B 0,C 180,E1 -17474.674,E2 -17474.674} C_VEL
LIN {X 0,Y 277.343,Z 192.936,A -85,B 0,C 180,E1 -17479.234,E2 -17479.234} C_VEL
LIN {X 0,Y 277.318,Z 192.942,A -85,B 0,C 180,E1 -17484.171,E2 -17484.171} C_VEL
LIN {X 0,Y 277.323,Z 192.942,A -85,B 0,C 180,E1 -17487.505,E2 -17487.505} C_VEL
LIN {X 0,Y 277.271,Z 192.945,A -85,B 0,C 180,E1 -17490.482,E2 -17490.482} C_VEL
LIN {X 0,Y 277.245,Z 192.95,A -85,B 0,C 180,E1 -17493.896,E2 -17493.896} C_VEL
LIN {X 0,Y 277.255,Z 192.95,A -85,B 0,C 180,E1 -17497.472,E2 -17497.472} C_VEL
LIN {X 0,Y 277.208,Z 192.958,A -85,B 0,C 180,E1 -17501.237,E2 -17501.237} C_VEL
LIN {X 0,Y 277.2,Z 192.957,A -85,B 0,C 180,E1 -17505.227,E2 -17505.227} C_VEL
LIN {X 0,Y 277.222,Z 192.955,A -85,B 0,C 180,E1 -17509.513,E2 -17509.513} C_VEL
LIN {X 0,Y 277.257,Z 193.247,A -85,B 0,C 180,E1 -17510.676,E2 -17510.676} C_VEL
LIN {X 0,Y 277.431,Z 196.101,A -85,B 0,C 180,E1 -17514.159,E2 -17514.159} C_VEL
LIN {X 0,Y 277.193,Z 199.326,A -85,B 0,C 180,E1 -17517.83,E2 -17517.83} C_VEL
LIN {X 0,Y 276.926,Z 202.431,A -85,B 0,C 180,E1 -17521.172,E2 -17521.172} C_VEL
LIN {X 0,Y 276.736,Z 204.612,A -85,B 0,C 180,E1 -17523.456,E2 -17523.456} C_VEL
LIN {X 0,Y 281.446,Z 219.795,A -85,B 0,C 180,E1 -17524.761,E2 -17524.761} C_VEL
LIN {X 0,Y 284.197,Z 231.161,A -85,B 0,C 180,E1 -17525.915,E2 -17525.915} C_VEL
LIN {X 0,Y 286.085,Z 242.413,A -85,B 0,C 180,E1 -17527.238,E2 -17527.238} C_VEL
LIN {X 0,Y 286.497,Z 245.545,A -85,B 0,C 180,E1 -17527.653,E2 -17527.653} C_VEL
LIN {X 0,Y 284.954,Z 256.581,A -85,B 0,C 180,E1 -17529.046,E2 -17529.046} C_VEL
LIN {X 0,Y 283.472,Z 265.649,A -85,B 0,C 180,E1 -17530.471,E2 -17530.471} C_VEL
LIN {X 0,Y 281.917,Z 274.679,A -85,B 0,C 180,E1 -17532.219,E2 -17532.219} C_VEL
LIN {X 0,Y 280.035,Z 283.587,A -85,B 0,C 180,E1 -17534.349,E2 -17534.349} C_VEL
LIN {X 0,Y 278.603,Z 290.752,A -85,B 0,C 180,E1 -17536.507,E2 -17536.507} C_VEL
LIN {X 0,Y 277.606,Z 295.582,A -85,B 0,C 180,E1 -17538.315,E2 -17538.315} C_VEL
LIN {X 0,Y 276.671,Z 300.275,A -85,B 0,C 180,E1 -17540.497,E2 -17540.497} C_VEL
LIN {X 0,Y 276.08,Z 303.863,A -85,B 0,C 180,E1 -17542.688,E2 -17542.688} C_VEL
LIN {X 0,Y 275.787,Z 305.716,A -85,B 0,C 180,E1 -17544.15,E2 -17544.15} C_VEL
LIN {X 0,Y 275.596,Z 307.109,A -85,B 0,C 180,E1 -17545.613,E2 -17545.613} C_VEL
LIN {X 0,Y 275.439,Z 308.1,A -85,B 0,C 180,E1 -17547.075,E2 -17547.075} C_VEL
LIN {X 0,Y 275.289,Z 308.941,A -85,B 0,C 180,E1 -17550,E2 -17550} C_VEL
LIN {X 0,Y 275.317,Z 308.748,A -85,B 0,C 180,E1 -17551.463,E2 -17551.463} C_VEL
LIN {X 0,Y 275.437,Z 308.161,A -85,B 0,C 180,E1 -17552.926,E2 -17552.926} C_VEL
LIN {X 0,Y 275.587,Z 307.194,A -85,B 0,C 180,E1 -17554.388,E2 -17554.388} C_VEL
LIN {X 0,Y 275.912,Z 304.97,A -85,B 0,C 180,E1 -17556.582,E2 -17556.582} C_VEL
LIN {X 0,Y 276.428,Z 301.778,A -85,B 0,C 180,E1 -17558.775,E2 -17558.775} C_VEL
LIN {X 0,Y 277.212,Z 297.527,A -85,B 0,C 180,E1 -17560.961,E2 -17560.961} C_VEL
LIN {X 0,Y 278.563,Z 291.087,A -85,B 0,C 180,E1 -17563.496,E2 -17563.496} C_VEL
LIN {X 0,Y 279.989,Z 284.008,A -85,B 0,C 180,E1 -17565.655,E2 -17565.655} C_VEL
LIN {X 0,Y 281.858,Z 275.184,A -85,B 0,C 180,E1 -17567.785,E2 -17567.785} C_VEL
LIN {X 0,Y 283.369,Z 266.299,A -85,B 0,C 180,E1 -17569.53,E2 -17569.53} C_VEL
LIN {X 0,Y 285.084,Z 256.102,A -85,B 0,C 180,E1 -17571.134,E2 -17571.134} C_VEL
LIN {X 0,Y 286.534,Z 246.517,A -85,B 0,C 180,E1 -17572.345,E2 -17572.345} C_VEL
LIN {X 0,Y 285.143,Z 236.246,A -85,B 0,C 180,E1 -17573.631,E2 -17573.631} C_VEL
LIN {X 0,Y 282.75,Z 224.774,A -85,B 0,C 180,E1 -17574.874,E2 -17574.874} C_VEL
LIN {X 0,Y 279.307,Z 212.686,A -85,B 0,C 180,E1 -17576.004,E2 -17576.004} C_VEL
LIN {X 0,Y 276.744,Z 204.611,A -85,B 0,C 180,E1 -17576.67,E2 -17576.67} C_VEL
LIN {X 0,Y 277.092,Z 200.989,A -85,B 0,C 180,E1 -17580.482,E2 -17580.482} C_VEL
LIN {X 0,Y 277.35,Z 197.951,A -85,B 0,C 180,E1 -17583.882,E2 -17583.882} C_VEL
LIN {X 0,Y 277.424,Z 194.88,A -85,B 0,C 180,E1 -17587.445,E2 -17587.445} C_VEL
LIN {X 0,Y 277.246,Z 193.36,A -85,B 0,C 180,E1 -17589.326,E2 -17589.326} C_VEL
LIN {X 0,Y 277.178,Z 192.957,A -85,B 0,C 180,E1 -17591.242,E2 -17591.242} C_VEL
LIN {X 0,Y 277.199,Z 192.956,A -85,B 0,C 180,E1 -17595.227,E2 -17595.227} C_VEL
LIN {X 0,Y 277.224,Z 192.953,A -85,B 0,C 180,E1 -17599.512,E2 -17599.512} C_VEL
LIN {X 0,Y 277.258,Z 192.95,A -85,B 0,C 180,E1 -17602.529,E2 -17602.529} C_VEL
LIN {X 0,Y 277.247,Z 192.949,A -85,B 0,C 180,E1 -17606.104,E2 -17606.104} C_VEL
LIN {X 0,Y 277.263,Z 192.946,A -85,B 0,C 180,E1 -17609.539,E2 -17609.539} C_VEL
LIN {X 0,Y 277.358,Z 192.935,A -85,B 0,C 180,E1 -17612.864,E2 -17612.864} C_VEL
LIN {X 0,Y 277.331,Z 192.941,A -85,B 0,C 180,E1 -17616.08,E2 -17616.08} C_VEL
LIN {X 0,Y 277.347,Z 192.935,A -85,B 0,C 180,E1 -17620.766,E2 -17620.766} C_VEL
LIN {X 0,Y 277.436,Z 192.926,A -85,B 0,C 180,E1 -17625.326,E2 -17625.326} C_VEL
LIN {X 0,Y 277.459,Z 192.924,A -85,B 0,C 180,E1 -17629.787,E2 -17629.787} C_VEL
LIN {X 0,Y 277.602,Z 192.904,A -85,B 0,C 180,E1 -17632.728,E2 -17632.728} C_VEL
LIN {X 0,Y 277.822,Z 192.877,A -85,B 0,C 180,E1 -17638.55,E2 -17638.55} C_VEL
LIN {X 0,Y 277.822,Z 192.879,A -85,B 0,C 180,E1 -17641.449,E2 -17641.449} C_VEL
LIN {X 0,Y 277.602,Z 192.906,A -85,B 0,C 180,E1 -17647.272,E2 -17647.272} C_VEL
LIN {X 0,Y 277.498,Z 192.917,A -85,B 0,C 180,E1 -17649.638,E2 -17649.638} C_VEL
LIN {X 0,Y 276.77,Z 193.012,A -85,B 0,C 180,E1 -17650.848,E2 -17650.848} C_VEL
LIN {X 0,Y 273.918,Z 193.368,A -85,B 0,C 180,E1 -17652.821,E2 -17652.821} C_VEL
LIN {X 0,Y 271.52,Z 193.666,A -85,B 0,C 180,E1 -17654.424,E2 -17654.424} C_VEL
LIN {X 0,Y 270.47,Z 193.795,A -85,B 0,C 180,E1 -17655.665,E2 -17655.665} C_VEL
LIN {X 0,Y 270.371,Z 193.807,A -85,B 0,C 180,E1 -17656.086,E2 -17656.086} C_VEL
LIN {X 0,Y 270.293,Z 193.818,A -85,B 0,C 180,E1 -17660.601,E2 -17660.601} C_VEL
LIN {X 0,Y 270.239,Z 193.823,A -85,B 0,C 180,E1 -17664.589,E2 -17664.589} C_VEL
LIN {X 0,Y 270.271,Z 193.821,A -85,B 0,C 180,E1 -17667.909,E2 -17667.909} C_VEL
LIN {X 0,Y 270.185,Z 193.832,A -85,B 0,C 180,E1 -17671.348,E2 -17671.348} C_VEL
LIN {X 0,Y 270.199,Z 193.829,A -85,B 0,C 180,E1 -17674.906,E2 -17674.906} C_VEL
LIN {X 0,Y 270.199,Z 193.829,A -85,B 0,C 180,E1 -17678.71,E2 -17678.71} C_VEL
LIN {X 0,Y 270.226,Z 193.946,A -85,B 0,C 180,E1 -17680.734,E2 -17680.734} C_VEL
LIN {X 0,Y 270.81,Z 197.491,A -85,B 0,C 180,E1 -17684.483,E2 -17684.483} C_VEL
LIN {X 0,Y 271.586,Z 201.717,A -85,B 0,C 180,E1 -17688.63,E2 -17688.63} C_VEL
LIN {X 0,Y 271.959,Z 205.043,A -85,B 0,C 180,E1 -17691.668,E2 -17691.668} C_VEL
LIN {X 0,Y 271.979,Z 208.245,A -85,B 0,C 180,E1 -17694.45,E2 -17694.45} C_VEL
LIN {X 0,Y 271.577,Z 211.44,A -85,B 0,C 180,E1 -17697.081,E2 -17697.081} C_VEL
LIN {X 0,Y 270.65,Z 216.682,A -85,B 0,C 180,E1 -17701.29,E2 -17701.29} C_VEL
LIN {X 0,Y 270.37,Z 218.461,A -85,B 0,C 180,E1 -17702.697,E2 -17702.697} C_VEL
LIN {X 0,Y 272.649,Z 227.242,A -85,B 0,C 180,E1 -17703.345,E2 -17703.345} C_VEL
LIN {X 0,Y 275.453,Z 240.132,A -85,B 0,C 180,E1 -17704.485,E2 -17704.485} C_VEL
LIN {X 0,Y 277.124,Z 251.54,A -85,B 0,C 180,E1 -17705.678,E2 -17705.678} C_VEL
LIN {X 0,Y 278.048,Z 262.37,A -85,B 0,C 180,E1 -17707.011,E2 -17707.011} C_VEL
LIN {X 0,Y 278.121,Z 268.909,A -85,B 0,C 180,E1 -17707.921,E2 -17707.921} C_VEL
LIN {X 0,Y 276.14,Z 279.56,A -85,B 0,C 180,E1 -17709.516,E2 -17709.516} C_VEL
LIN {X 0,Y 274.364,Z 289.033,A -85,B 0,C 180,E1 -17711.296,E2 -17711.296} C_VEL
LIN {X 0,Y 272.812,Z 297.039,A -85,B 0,C 180,E1 -17713.153,E2 -17713.153} C_VEL
LIN {X 0,Y 271.226,Z 304.731,A -85,B 0,C 180,E1 -17715.366,E2 -17715.366} C_VEL
LIN {X 0,Y 269.821,Z 311.828,A -85,B 0,C 180,E1 -17717.973,E2 -17717.973} C_VEL
LIN {X 0,Y 269.015,Z 316.553,A -85,B 0,C 180,E1 -17720.223,E2 -17720.223} C_VEL
LIN {X 0,Y 268.498,Z 320.165,A -85,B 0,C 180,E1 -17722.479,E2 -17722.479} C_VEL
LIN {X 0,Y 268.212,Z 322.729,A -85,B 0,C 180,E1 -17724.698,E2 -17724.698} C_VEL
LIN {X 0,Y 268.173,Z 324.429,A -85,B 0,C 180,E1 -17726.995,E2 -17726.995} C_VEL
LIN {X 0,Y 268.179,Z 325.039,A -85,B 0,C 180,E1 -17728.498,E2 -17728.498} C_VEL
LIN {X 0,Y 268.176,Z 325.254,A -85,B 0,C 180,E1 -17730,E2 -17730} C_VEL
LIN {X 0,Y 268.179,Z 325.034,A -85,B 0,C 180,E1 -17731.501,E2 -17731.501} C_VEL
LIN {X 0,Y 268.173,Z 324.42,A -85,B 0,C 180,E1 -17733.004,E2 -17733.004} C_VEL
LIN {X 0,Y 268.226,Z 322.682,A -85,B 0,C 180,E1 -17735.334,E2 -17735.334} C_VEL
LIN {X 0,Y 268.64,Z 319.064,A -85,B 0,C 180,E1 -17738.272,E2 -17738.272} C_VEL
LIN {X 0,Y 269.258,Z 315.079,A -85,B 0,C 180,E1 -17740.527,E2 -17740.527} C_VEL
LIN {X 0,Y 270.325,Z 308.953,A -85,B 0,C 180,E1 -17743.149,E2 -17743.149} C_VEL
LIN {X 0,Y 271.754,Z 302.269,A -85,B 0,C 180,E1 -17745.371,E2 -17745.371} C_VEL
LIN {X 0,Y 273.481,Z 293.979,A -85,B 0,C 180,E1 -17747.575,E2 -17747.575} C_VEL
LIN {X 0,Y 274.988,Z 285.474,A -85,B 0,C 180,E1 -17749.405,E2 -17749.405} C_VEL
LIN {X 0,Y 276.956,Z 274.976,A -85,B 0,C 180,E1 -17751.198,E2 -17751.198} C_VEL
LIN {X 0,Y 278.207,Z 267.442,A -85,B 0,C 180,E1 -17752.267,E2 -17752.267} C_VEL
LIN {X 0,Y 277.625,Z 256.435,A -85,B 0,C 180,E1 -17753.72,E2 -17753.72} C_VEL
LIN {X 0,Y 276.167,Z 244.189,A -85,B 0,C 180,E1 -17755.083,E2 -17755.083} C_VEL
LIN {X 0,Y 273.705,Z 231.568,A -85,B 0,C 180,E1 -17756.272,E2 -17756.272} C_VEL
LIN {X 0,Y 270.372,Z 218.445,A -85,B 0,C 180,E1 -17757.29,E2 -17757.29} C_VEL
LIN {X 0,Y 271.193,Z 213.521,A -85,B 0,C 180,E1 -17761.218,E2 -17761.218} C_VEL
LIN {X 0,Y 271.96,Z 209.287,A -85,B 0,C 180,E1 -17764.647,E2 -17764.647} C_VEL
LIN {X 0,Y 272.054,Z 206.76,A -85,B 0,C 180,E1 -17766.791,E2 -17766.791} C_VEL
LIN {X 0,Y 271.78,Z 202.857,A -85,B 0,C 180,E1 -17770.276,E2 -17770.276} C_VEL
LIN {X 0,Y 270.984,Z 198.529,A -85,B 0,C 180,E1 -17774.446,E2 -17774.446} C_VEL
LIN {X 0,Y 270.492,Z 195.542,A -85,B 0,C 180,E1 -17777.504,E2 -17777.504} C_VEL
LIN {X 0,Y 270.196,Z 193.831,A -85,B 0,C 180,E1 -17779.438,E2 -17779.438} C_VEL
LIN {X 0,Y 270.218,Z 193.827,A -85,B 0,C 180,E1 -17783.732,E2 -17783.732} C_VEL
LIN {X 0,Y 270.201,Z 193.828,A -85,B 0,C 180,E1 -17786.892,E2 -17786.892} C_VEL
LIN {X 0,Y 270.194,Z 193.829,A -85,B 0,C 180,E1 -17790.382,E2 -17790.382} C_VEL
LIN {X 0,Y 270.259,Z 193.823,A -85,B 0,C 180,E1 -17793.763,E2 -17793.763} C_VEL
LIN {X 0,Y 270.209,Z 193.827,A -85,B 0,C 180,E1 -17797.037,E2 -17797.037} C_VEL
LIN {X 0,Y 270.299,Z 193.816,A -85,B 0,C 180,E1 -17800.244,E2 -17800.244} C_VEL
LIN {X 0,Y 270.401,Z 193.802,A -85,B 0,C 180,E1 -17804.935,E2 -17804.935} C_VEL
LIN {X 0,Y 270.408,Z 193.799,A -85,B 0,C 180,E1 -17809.518,E2 -17809.518} C_VEL
LIN {X 0,Y 270.56,Z 193.782,A -85,B 0,C 180,E1 -17812.537,E2 -17812.537} C_VEL
LIN {X 0,Y 270.784,Z 193.754,A -85,B 0,C 180,E1 -17818.513,E2 -17818.513} C_VEL
LIN {X 0,Y 270.784,Z 193.753,A -85,B 0,C 180,E1 -17821.487,E2 -17821.487} C_VEL
LIN {X 0,Y 270.56,Z 193.78,A -85,B 0,C 180,E1 -17827.463,E2 -17827.463} C_VEL
LIN {X 0,Y 270.408,Z 193.803,A -85,B 0,C 180,E1 -17830.482,E2 -17830.482} C_VEL
LIN {X 0,Y 270.401,Z 193.8,A -85,B 0,C 180,E1 -17835.065,E2 -17835.065} C_VEL
LIN {X 0,Y 270.3,Z 193.816,A -85,B 0,C 180,E1 -17839.756,E2 -17839.756} C_VEL
LIN {X 0,Y 270.273,Z 193.817,A -85,B 0,C 180,E1 -17844.586,E2 -17844.586} C_VEL
LIN {X 0,Y 270.269,Z 193.821,A -85,B 0,C 180,E1 -17847.909,E2 -17847.909} C_VEL
LIN {X 0,Y 270.183,Z 193.831,A -85,B 0,C 180,E1 -17851.349,E2 -17851.349} C_VEL
LIN {X 0,Y 270.197,Z 193.829,A -85,B 0,C 180,E1 -17854.906,E2 -17854.906} C_VEL
LIN {X 0,Y 270.196,Z 193.83,A -85,B 0,C 180,E1 -17858.711,E2 -17858.711} C_VEL
LIN {X 0,Y 270.164,Z 193.835,A -85,B 0,C 180,E1 -17863.249,E2 -17863.249} C_VEL
LIN {X 0,Y 270.171,Z 193.833,A -85,B 0,C 180,E1 -17867.442,E2 -17867.442} C_VEL
LIN {X 0,Y 270.173,Z 193.833,A -85,B 0,C 180,E1 -17869.435,E2 -17869.435} C_VEL
LIN {X 0,Y 270.314,Z 194.969,A -85,B 0,C 180,E1 -17871.393,E2 -17871.393} C_VEL
LIN {X 0,Y 270.413,Z 196.805,A -85,B 0,C 180,E1 -17873.677,E2 -17873.677} C_VEL
LIN {X 0,Y 270.247,Z 199.546,A -85,B 0,C 180,E1 -17876.899,E2 -17876.899} C_VEL
LIN {X 0,Y 269.964,Z 202.649,A -85,B 0,C 180,E1 -17880.355,E2 -17880.355} C_VEL
LIN {X 0,Y 269.776,Z 205.047,A -85,B 0,C 180,E1 -17882.746,E2 -17882.746} C_VEL
LIN {X 0,Y 274.035,Z 218.153,A -85,B 0,C 180,E1 -17883.9,E2 -17883.9} C_VEL
LIN {X 0,Y 277.008,Z 229.699,A -85,B 0,C 180,E1 -17885.096,E2 -17885.096} C_VEL
LIN {X 0,Y 279.079,Z 241.382,A -85,B 0,C 180,E1 -17886.488,E2 -17886.488} C_VEL
LIN {X 0,Y 279.824,Z 247.338,A -85,B 0,C 180,E1 -17887.286,E2 -17887.286} C_VEL
LIN {X 0,Y 278.13,Z 257.982,A -85,B 0,C 180,E1 -17888.701,E2 -17888.701} C_VEL
LIN {X 0,Y 276.462,Z 267.829,A -85,B 0,C 180,E1 -17890.345,E2 -17890.345} C_VEL
LIN {X 0,Y 274.826,Z 276.515,A -85,B 0,C 180,E1 -17892.13,E2 -17892.13} C_VEL
LIN {X 0,Y 272.942,Z 285.13,A -85,B 0,C 180,E1 -17894.314,E2 -17894.314} C_VEL
LIN {X 0,Y 271.474,Z 291.994,A -85,B 0,C 180,E1 -17896.527,E2 -17896.527} C_VEL
LIN {X 0,Y 270.274,Z 297.488,A -85,B 0,C 180,E1 -17898.754,E2 -17898.754} C_VEL
LIN {X 0,Y 269.442,Z 301.798,A -85,B 0,C 180,E1 -17900.997,E2 -17900.997} C_VEL
LIN {X 0,Y 268.849,Z 305.225,A -85,B 0,C 180,E1 -17903.397,E2 -17903.397} C_VEL
LIN {X 0,Y 268.525,Z 307.322,A -85,B 0,C 180,E1 -17905.497,E2 -17905.497} C_VEL
LIN {X 0,Y 268.375,Z 308.313,A -85,B 0,C 180,E1 -17906.998,E2 -17906.998} C_VEL
LIN {X 0,Y 268.213,Z 309.154,A -85,B 0,C 180,E1 -17910,E2 -17910} C_VEL
LIN {X 0,Y 268.245,Z 308.96,A -85,B 0,C 180,E1 -17911.502,E2 -17911.502} C_VEL
LIN {X 0,Y 268.373,Z 308.373,A -85,B 0,C 180,E1 -17913.003,E2 -17913.003} C_VEL
LIN {X 0,Y 268.516,Z 307.406,A -85,B 0,C 180,E1 -17914.504,E2 -17914.504} C_VEL
LIN {X 0,Y 268.795,Z 305.481,A -85,B 0,C 180,E1 -17916.503,E2 -17916.503} C_VEL
LIN {X 0,Y 269.409,Z 301.99,A -85,B 0,C 180,E1 -17919.005,E2 -17919.005} C_VEL
LIN {X 0,Y 270.234,Z 297.739,A -85,B 0,C 180,E1 -17921.248,E2 -17921.248} C_VEL
LIN {X 0,Y 271.679,Z 291.298,A -85,B 0,C 180,E1 -17923.845,E2 -17923.845} C_VEL
LIN {X 0,Y 273.156,Z 284.219,A -85,B 0,C 180,E1 -17926.057,E2 -17926.057} C_VEL
LIN {X 0,Y 275.116,Z 275.394,A -85,B 0,C 180,E1 -17928.236,E2 -17928.236} C_VEL
LIN {X 0,Y 276.798,Z 266.053,A -85,B 0,C 180,E1 -17930.104,E2 -17930.104} C_VEL
LIN {X 0,Y 278.484,Z 256.31,A -85,B 0,C 180,E1 -17931.66,E2 -17931.66} C_VEL
LIN {X 0,Y 279.808,Z 248.208,A -85,B 0,C 180,E1 -17932.717,E2 -17932.717} C_VEL
LIN {X 0,Y 278.718,Z 238.815,A -85,B 0,C 180,E1 -17933.956,E2 -17933.956} C_VEL
LIN {X 0,Y 276.449,Z 227.259,A -85,B 0,C 180,E1 -17935.301,E2 -17935.301} C_VEL
LIN {X 0,Y 273.005,Z 214.874,A -85,B 0,C 180,E1 -17936.538,E2 -17936.538} C_VEL
LIN {X 0,Y 269.827,Z 205.357,A -85,B 0,C 180,E1 -17937.362,E2 -17937.362} C_VEL
LIN {X 0,Y 269.734,Z 204.852,A -85,B 0,C 180,E1 -17937.413,E2 -17937.413} C_VEL
LIN {X 0,Y 270.103,Z 201.206,A -85,B 0,C 180,E1 -17941.359,E2 -17941.359} C_VEL
LIN {X 0,Y 270.364,Z 198.147,A -85,B 0,C 180,E1 -17944.882,E2 -17944.882} C_VEL
LIN {X 0,Y 270.416,Z 196.609,A -85,B 0,C 180,E1 -17946.71,E2 -17946.71} C_VEL
LIN {X 0,Y 270.311,Z 194.979,A -85,B 0,C 180,E1 -17948.74,E2 -17948.74} C_VEL
LIN {X 0,Y 270.131,Z 193.834,A -85,B 0,C 180,E1 -17950.574,E2 -17950.574} C_VEL
LIN {X 0,Y 270.147,Z 193.833,A -85,B 0,C 180,E1 -17954.621,E2 -17954.621} C_VEL
LIN {X 0,Y 270.173,Z 193.831,A -85,B 0,C 180,E1 -17957.442,E2 -17957.442} C_VEL
LIN {X 0,Y 270.209,Z 193.827,A -85,B 0,C 180,E1 -17961.374,E2 -17961.374} C_VEL
LIN {X 0,Y 270.199,Z 193.828,A -85,B 0,C 180,E1 -17965.094,E2 -17965.094} C_VEL
LIN {X 0,Y 270.202,Z 193.827,A -85,B 0,C 180,E1 -17969.131,E2 -17969.131} C_VEL
LIN {X 0,Y 270.265,Z 193.82,A -85,B 0,C 180,E1 -17972.146,E2 -17972.146} C_VEL
LIN {X 0,Y 270.279,Z 193.816,A -85,B 0,C 180,E1 -17975.519,E2 -17975.519} C_VEL
LIN {X 0,Y 270.303,Z 193.815,A -85,B 0,C 180,E1 -17980.244,E2 -17980.244} C_VEL
LIN {X 0,Y 270.405,Z 193.801,A -85,B 0,C 180,E1 -17984.935,E2 -17984.935} C_VEL
LIN {X 0,Y 270.411,Z 193.803,A -85,B 0,C 180,E1 -17989.518,E2 -17989.518} C_VEL
LIN {X 0,Y 270.564,Z 193.78,A -85,B 0,C 180,E1 -17992.537,E2 -17992.537} C_VEL
LIN {X 0,Y 270.787,Z 193.753,A -85,B 0,C 180,E1 -17998.513,E2 -17998.513} C_VEL
LIN {X 0,Y 270.788,Z 193.755,A -85,B 0,C 180,E1 -18001.487,E2 -18001.487} C_VEL
LIN {X 0,Y 270.564,Z 193.782,A -85,B 0,C 180,E1 -18007.462,E2 -18007.462} C_VEL
LIN {X 0,Y 270.414,Z 193.802,A -85,B 0,C 180,E1 -18010.482,E2 -18010.482} C_VEL
LIN {X 0,Y 270.405,Z 193.803,A -85,B 0,C 180,E1 -18015.065,E2 -18015.065} C_VEL
LIN {X 0,Y 270.371,Z 193.807,A -85,B 0,C 180,E1 -18016.086,E2 -18016.086} C_VEL
LIN {X 0,Y 269.649,Z 193.898,A -85,B 0,C 180,E1 -18017.33,E2 -18017.33} C_VEL
LIN {X 0,Y 266.717,Z 194.264,A -85,B 0,C 180,E1 -18019.354,E2 -18019.354} C_VEL
LIN {X 0,Y 264.255,Z 194.569,A -85,B 0,C 180,E1 -18021.001,E2 -18021.001} C_VEL
LIN {X 0,Y 263.206,Z 194.7,A -85,B 0,C 180,E1 -18022.279,E2 -18022.279} C_VEL
LIN {X 0,Y 263.124,Z 194.706,A -85,B 0,C 180,E1 -18022.712,E2 -18022.712} C_VEL
LIN {X 0,Y 263.194,Z 194.7,A -85,B 0,C 180,E1 -18025.293,E2 -18025.293} C_VEL
LIN {X 0,Y 263.167,Z 194.704,A -85,B 0,C 180,E1 -18028.731,E2 -18028.731} C_VEL
LIN {X 0,Y 263.134,Z 194.711,A -85,B 0,C 180,E1 -18032.288,E2 -18032.288} C_VEL
LIN {X 0,Y 263.177,Z 194.704,A -85,B 0,C 180,E1 -18036.761,E2 -18036.761} C_VEL
LIN {X 0,Y 263.144,Z 194.816,A -85,B 0,C 180,E1 -18040.115,E2 -18040.115} C_VEL
LIN {X 0,Y 263.769,Z 198.354,A -85,B 0,C 180,E1 -18043.995,E2 -18043.995} C_VEL
LIN {X 0,Y 264.549,Z 202.681,A -85,B 0,C 180,E1 -18048.383,E2 -18048.383} C_VEL
LIN {X 0,Y 264.936,Z 205.897,A -85,B 0,C 180,E1 -18051.436,E2 -18051.436} C_VEL
LIN {X 0,Y 264.903,Z 210.295,A -85,B 0,C 180,E1 -18055.33,E2 -18055.33} C_VEL
LIN {X 0,Y 263.94,Z 215.417,A -85,B 0,C 180,E1 -18059.607,E2 -18059.607} C_VEL
LIN {X 0,Y 263.475,Z 218.247,A -85,B 0,C 180,E1 -18061.921,E2 -18061.921} C_VEL
LIN {X 0,Y 265.73,Z 226.916,A -85,B 0,C 180,E1 -18062.587,E2 -18062.587} C_VEL
LIN {X 0,Y 268.487,Z 239.062,A -85,B 0,C 180,E1 -18063.705,E2 -18063.705} C_VEL
LIN {X 0,Y 270.228,Z 250.174,A -85,B 0,C 180,E1 -18064.898,E2 -18064.898} C_VEL
LIN {X 0,Y 271.227,Z 261.328,A -85,B 0,C 180,E1 -18066.293,E2 -18066.293} C_VEL
LIN {X 0,Y 271.508,Z 268.698,A -85,B 0,C 180,E1 -18067.354,E2 -18067.354} C_VEL
LIN {X 0,Y 269.488,Z 279.35,A -85,B 0,C 180,E1 -18068.986,E2 -18068.986} C_VEL
LIN {X 0,Y 267.539,Z 289.235,A -85,B 0,C 180,E1 -18070.894,E2 -18070.894} C_VEL
LIN {X 0,Y 266.01,Z 296.828,A -85,B 0,C 180,E1 -18072.709,E2 -18072.709} C_VEL
LIN {X 0,Y 264.334,Z 304.518,A -85,B 0,C 180,E1 -18074.975,E2 -18074.975} C_VEL
LIN {X 0,Y 262.827,Z 311.614,A -85,B 0,C 180,E1 -18077.647,E2 -18077.647} C_VEL
LIN {X 0,Y 262.007,Z 316.34,A -85,B 0,C 180,E1 -18079.959,E2 -18079.959} C_VEL
LIN {X 0,Y 261.428,Z 319.952,A -85,B 0,C 180,E1 -18082.275,E2 -18082.275} C_VEL
LIN {X 0,Y 261.124,Z 322.721,A -85,B 0,C 180,E1 -18084.769,E2 -18084.769} C_VEL
LIN {X 0,Y 261.089,Z 324.216,A -85,B 0,C 180,E1 -18086.914,E2 -18086.914} C_VEL
LIN {X 0,Y 261.107,Z 324.827,A -85,B 0,C 180,E1 -18088.457,E2 -18088.457} C_VEL
LIN {X 0,Y 261.103,Z 325.042,A -85,B 0,C 180,E1 -18090,E2 -18090} C_VEL
LIN {X 0,Y 261.107,Z 324.821,A -85,B 0,C 180,E1 -18091.542,E2 -18091.542} C_VEL
LIN {X 0,Y 261.089,Z 324.207,A -85,B 0,C 180,E1 -18093.086,E2 -18093.086} C_VEL
LIN {X 0,Y 261.231,Z 321.799,A -85,B 0,C 180,E1 -18096.177,E2 -18096.177} C_VEL
LIN {X 0,Y 261.588,Z 318.85,A -85,B 0,C 180,E1 -18098.497,E2 -18098.497} C_VEL
LIN {X 0,Y 262.252,Z 314.864,A -85,B 0,C 180,E1 -18100.812,E2 -18100.812} C_VEL
LIN {X 0,Y 263.393,Z 308.737,A -85,B 0,C 180,E1 -18103.501,E2 -18103.501} C_VEL
LIN {X 0,Y 264.902,Z 302.054,A -85,B 0,C 180,E1 -18105.779,E2 -18105.779} C_VEL
LIN {X 0,Y 266.7,Z 293.763,A -85,B 0,C 180,E1 -18108.037,E2 -18108.037} C_VEL
LIN {X 0,Y 268.263,Z 285.257,A -85,B 0,C 180,E1 -18109.912,E2 -18109.912} C_VEL
LIN {X 0,Y 270.342,Z 274.758,A -85,B 0,C 180,E1 -18111.743,E2 -18111.743} C_VEL
LIN {X 0,Y 271.435,Z 268.545,A -85,B 0,C 180,E1 -18112.652,E2 -18112.652} C_VEL
LIN {X 0,Y 270.915,Z 257.288,A -85,B 0,C 180,E1 -18114.221,E2 -18114.221} C_VEL
LIN {X 0,Y 269.475,Z 244.812,A -85,B 0,C 180,E1 -18115.673,E2 -18115.673} C_VEL
LIN {X 0,Y 266.973,Z 231.848,A -85,B 0,C 180,E1 -18116.952,E2 -18116.952} C_VEL
LIN {X 0,Y 263.443,Z 218.235,A -85,B 0,C 180,E1 -18118.064,E2 -18118.064} C_VEL
LIN {X 0,Y 264.311,Z 213.304,A -85,B 0,C 180,E1 -18122.126,E2 -18122.126} C_VEL
LIN {X 0,Y 264.903,Z 210.258,A -85,B 0,C 180,E1 -18124.67,E2 -18124.67} C_VEL
LIN {X 0,Y 265.004,Z 206.939,A -85,B 0,C 180,E1 -18127.587,E2 -18127.587} C_VEL
LIN {X 0,Y 264.744,Z 203.718,A -85,B 0,C 180,E1 -18130.569,E2 -18130.569} C_VEL
LIN {X 0,Y 264.07,Z 200.19,A -85,B 0,C 180,E1 -18134.062,E2 -18134.062} C_VEL
LIN {X 0,Y 263.4,Z 196.156,A -85,B 0,C 180,E1 -18138.338,E2 -18138.338} C_VEL
LIN {X 0,Y 263.118,Z 194.709,A -85,B 0,C 180,E1 -18140.13,E2 -18140.13} C_VEL
LIN {X 0,Y 263.156,Z 194.707,A -85,B 0,C 180,E1 -18144.017,E2 -18144.017} C_VEL
LIN {X 0,Y 263.131,Z 194.709,A -85,B 0,C 180,E1 -18147.711,E2 -18147.711} C_VEL
LIN {X 0,Y 263.194,Z 194.702,A -85,B 0,C 180,E1 -18151.785,E2 -18151.785} C_VEL
LIN {X 0,Y 263.199,Z 194.701,A -85,B 0,C 180,E1 -18155.212,E2 -18155.212} C_VEL
LIN {X 0,Y 263.261,Z 194.694,A -85,B 0,C 180,E1 -18159.693,E2 -18159.693} C_VEL
LIN {X 0,Y 263.349,Z 194.68,A -85,B 0,C 180,E1 -18164.522,E2 -18164.522} C_VEL
LIN {X 0,Y 263.351,Z 194.678,A -85,B 0,C 180,E1 -18169.233,E2 -18169.233} C_VEL
LIN {X 0,Y 263.524,Z 194.658,A -85,B 0,C 180,E1 -18172.337,E2 -18172.337} C_VEL
LIN {X 0,Y 263.749,Z 194.63,A -85,B 0,C 180,E1 -18178.473,E2 -18178.473} C_VEL
LIN {X 0,Y 263.748,Z 194.63,A -85,B 0,C 180,E1 -18181.527,E2 -18181.527} C_VEL
LIN {X 0,Y 263.524,Z 194.657,A -85,B 0,C 180,E1 -18187.663,E2 -18187.663} C_VEL
LIN {X 0,Y 263.351,Z 194.681,A -85,B 0,C 180,E1 -18190.767,E2 -18190.767} C_VEL
LIN {X 0,Y 263.349,Z 194.679,A -85,B 0,C 180,E1 -18195.478,E2 -18195.478} C_VEL
LIN {X 0,Y 263.262,Z 194.691,A -85,B 0,C 180,E1 -18200.307,E2 -18200.307} C_VEL
LIN {X 0,Y 263.207,Z 194.699,A -85,B 0,C 180,E1 -18205.292,E2 -18205.292} C_VEL
LIN {X 0,Y 263.175,Z 194.702,A -85,B 0,C 180,E1 -18208.73,E2 -18208.73} C_VEL
LIN {X 0,Y 263.132,Z 194.707,A -85,B 0,C 180,E1 -18212.289,E2 -18212.289} C_VEL
LIN {X 0,Y 263.175,Z 194.703,A -85,B 0,C 180,E1 -18216.762,E2 -18216.762} C_VEL
LIN {X 0,Y 263.104,Z 194.712,A -85,B 0,C 180,E1 -18219.873,E2 -18219.873} C_VEL
LIN {X 0,Y 263.103,Z 194.712,A -85,B 0,C 180,E1 -18223.989,E2 -18223.989} C_VEL
LIN {X 0,Y 263.124,Z 194.711,A -85,B 0,C 180,E1 -18228.407,E2 -18228.407} C_VEL
LIN {X 0,Y 263.169,Z 195.185,A -85,B 0,C 180,E1 -18230.14,E2 -18230.14} C_VEL
LIN {X 0,Y 263.386,Z 198.231,A -85,B 0,C 180,E1 -18234.054,E2 -18234.054} C_VEL
LIN {X 0,Y 263.121,Z 201.309,A -85,B 0,C 180,E1 -18237.711,E2 -18237.711} C_VEL
LIN {X 0,Y 262.761,Z 204.84,A -85,B 0,C 180,E1 -18241.675,E2 -18241.675} C_VEL
LIN {X 0,Y 262.783,Z 205.224,A -85,B 0,C 180,E1 -18241.954,E2 -18241.954} C_VEL
LIN {X 0,Y 264.828,Z 211.212,A -85,B 0,C 180,E1 -18242.473,E2 -18242.473} C_VEL
LIN {X 0,Y 268.528,Z 223.384,A -85,B 0,C 180,E1 -18243.688,E2 -18243.688} C_VEL
LIN {X 0,Y 270.967,Z 233.741,A -85,B 0,C 180,E1 -18244.868,E2 -18244.868} C_VEL
LIN {X 0,Y 272.719,Z 244.937,A -85,B 0,C 180,E1 -18246.32,E2 -18246.32} C_VEL
LIN {X 0,Y 273.051,Z 249.161,A -85,B 0,C 180,E1 -18246.915,E2 -18246.915} C_VEL
LIN {X 0,Y 271.091,Z 260.539,A -85,B 0,C 180,E1 -18248.52,E2 -18248.52} C_VEL
LIN {X 0,Y 269.478,Z 269.845,A -85,B 0,C 180,E1 -18250.182,E2 -18250.182} C_VEL
LIN {X 0,Y 267.727,Z 278.325,A -85,B 0,C 180,E1 -18252.035,E2 -18252.035} C_VEL
LIN {X 0,Y 265.831,Z 286.571,A -85,B 0,C 180,E1 -18254.277,E2 -18254.277} C_VEL
LIN {X 0,Y 264.586,Z 292.208,A -85,B 0,C 180,E1 -18256.169,E2 -18256.169} C_VEL
LIN {X 0,Y 263.308,Z 297.703,A -85,B 0,C 180,E1 -18258.453,E2 -18258.453} C_VEL
LIN {X 0,Y 262.409,Z 302.013,A -85,B 0,C 180,E1 -18260.753,E2 -18260.753} C_VEL
LIN {X 0,Y 261.727,Z 305.748,A -85,B 0,C 180,E1 -18263.486,E2 -18263.486} C_VEL
LIN {X 0,Y 261.457,Z 307.536,A -85,B 0,C 180,E1 -18265.375,E2 -18265.375} C_VEL
LIN {X 0,Y 261.29,Z 308.526,A -85,B 0,C 180,E1 -18266.917,E2 -18266.917} C_VEL
LIN {X 0,Y 261.139,Z 309.366,A -85,B 0,C 180,E1 -18270,E2 -18270} C_VEL
LIN {X 0,Y 261.174,Z 309.172,A -85,B 0,C 180,E1 -18271.542,E2 -18271.542} C_VEL
LIN {X 0,Y 261.289,Z 308.586,A -85,B 0,C 180,E1 -18273.084,E2 -18273.084} C_VEL
LIN {X 0,Y 261.449,Z 307.619,A -85,B 0,C 180,E1 -18274.626,E2 -18274.626} C_VEL
LIN {X 0,Y 261.727,Z 305.881,A -85,B 0,C 180,E1 -18276.514,E2 -18276.514} C_VEL
LIN {X 0,Y 262.379,Z 302.203,A -85,B 0,C 180,E1 -18279.249,E2 -18279.249} C_VEL
LIN {X 0,Y 263.272,Z 297.951,A -85,B 0,C 180,E1 -18281.55,E2 -18281.55} C_VEL
LIN {X 0,Y 264.801,Z 291.509,A -85,B 0,C 180,E1 -18284.212,E2 -18284.212} C_VEL
LIN {X 0,Y 266.342,Z 284.43,A -85,B 0,C 180,E1 -18286.479,E2 -18286.479} C_VEL
LIN {X 0,Y 268.376,Z 275.605,A -85,B 0,C 180,E1 -18288.711,E2 -18288.711} C_VEL
LIN {X 0,Y 270.144,Z 266.203,A -85,B 0,C 180,E1 -18290.633,E2 -18290.633} C_VEL
LIN {X 0,Y 271.887,Z 256.519,A -85,B 0,C 180,E1 -18292.213,E2 -18292.213} C_VEL
LIN {X 0,Y 273.155,Z 248.525,A -85,B 0,C 180,E1 -18293.288,E2 -18293.288} C_VEL
LIN {X 0,Y 271.836,Z 238.349,A -85,B 0,C 180,E1 -18294.682,E2 -18294.682} C_VEL
LIN {X 0,Y 269.425,Z 226.619,A -85,B 0,C 180,E1 -18296.081,E2 -18296.081} C_VEL
LIN {X 0,Y 265.72,Z 213.793,A -85,B 0,C 180,E1 -18297.402,E2 -18297.402} C_VEL
LIN {X 0,Y 262.85,Z 205.568,A -85,B 0,C 180,E1 -18298.152,E2 -18298.152} C_VEL
LIN {X 0,Y 262.773,Z 205.069,A -85,B 0,C 180,E1 -18298.2,E2 -18298.2} C_VEL
LIN {X 0,Y 263.127,Z 201.424,A -85,B 0,C 180,E1 -18302.289,E2 -18302.289} C_VEL
LIN {X 0,Y 263.324,Z 199.815,A -85,B 0,C 180,E1 -18304.17,E2 -18304.17} C_VEL
LIN {X 0,Y 263.326,Z 196.814,A -85,B 0,C 180,E1 -18307.869,E2 -18307.869} C_VEL
LIN {X 0,Y 263.169,Z 195.305,A -85,B 0,C 180,E1 -18309.861,E2 -18309.861} C_VEL
LIN {X 0,Y 263.077,Z 194.713,A -85,B 0,C 180,E1 -18311.903,E2 -18311.903} C_VEL
LIN {X 0,Y 263.106,Z 194.71,A -85,B 0,C 180,E1 -18316.155,E2 -18316.155} C_VEL
LIN {X 0,Y 263.107,Z 194.711,A -85,B 0,C 180,E1 -18320.127,E2 -18320.127} C_VEL
LIN {X 0,Y 263.159,Z 194.704,A -85,B 0,C 180,E1 -18324.017,E2 -18324.017} C_VEL
LIN {X 0,Y 263.134,Z 194.705,A -85,B 0,C 180,E1 -18327.712,E2 -18327.712} C_VEL
LIN {X 0,Y 263.198,Z 194.699,A -85,B 0,C 180,E1 -18331.785,E2 -18331.785} C_VEL
LIN {X 0,Y 263.228,Z 194.694,A -85,B 0,C 180,E1 -18335.2,E2 -18335.2} C_VEL
LIN {X 0,Y 263.265,Z 194.691,A -85,B 0,C 180,E1 -18339.693,E2 -18339.693} C_VEL
LIN {X 0,Y 263.353,Z 194.68,A -85,B 0,C 180,E1 -18344.522,E2 -18344.522} C_VEL
LIN {X 0,Y 263.354,Z 194.68,A -85,B 0,C 180,E1 -18349.233,E2 -18349.233} C_VEL
LIN {X 0,Y 263.528,Z 194.657,A -85,B 0,C 180,E1 -18352.337,E2 -18352.337} C_VEL
LIN {X 0,Y 263.751,Z 194.629,A -85,B 0,C 180,E1 -18358.473,E2 -18358.473} C_VEL
LIN {X 0,Y 263.752,Z 194.631,A -85,B 0,C 180,E1 -18361.527,E2 -18361.527} C_VEL
LIN {X 0,Y 263.527,Z 194.658,A -85,B 0,C 180,E1 -18367.663,E2 -18367.663} C_VEL
LIN {X 0,Y 263.357,Z 194.684,A -85,B 0,C 180,E1 -18370.766,E2 -18370.766} C_VEL
LIN {X 0,Y 263.353,Z 194.681,A -85,B 0,C 180,E1 -18375.478,E2 -18375.478} C_VEL
LIN {X 0,Y 263.264,Z 194.693,A -85,B 0,C 180,E1 -18380.307,E2 -18380.307} C_VEL
LIN {X 0,Y 263.124,Z 194.706,A -85,B 0,C 180,E1 -18382.712,E2 -18382.712} C_VEL
LIN {X 0,Y 262.463,Z 194.793,A -85,B 0,C 180,E1 -18383.989,E2 -18383.989} C_VEL
LIN {X 0,Y 259.616,Z 195.148,A -85,B 0,C 180,E1 -18386.071,E2 -18386.071} C_VEL
LIN {X 0,Y 257.204,Z 195.448,A -85,B 0,C 180,E1 -18387.764,E2 -18387.764} C_VEL
LIN {X 0,Y 256.181,Z 195.574,A -85,B 0,C 180,E1 -18389.077,E2 -18389.077} C_VEL
LIN {X 0,Y 256.104,Z 195.585,A -85,B 0,C 180,E1 -18389.522,E2 -18389.522} C_VEL
LIN {X 0,Y 256.069,Z 195.592,A -85,B 0,C 180,E1 -18393.293,E2 -18393.293} C_VEL
LIN {X 0,Y 256.111,Z 195.585,A -85,B 0,C 180,E1 -18397.269,E2 -18397.269} C_VEL
LIN {X 0,Y 256.109,Z 195.688,A -85,B 0,C 180,E1 -18399.475,E2 -18399.475} C_VEL
LIN {X 0,Y 256.646,Z 198.965,A -85,B 0,C 180,E1 -18403.204,E2 -18403.204} C_VEL
LIN {X 0,Y 257.372,Z 203.02,A -85,B 0,C 180,E1 -18407.501,E2 -18407.501} C_VEL
LIN {X 0,Y 257.784,Z 205.265,A -85,B 0,C 180,E1 -18409.762,E2 -18409.762} C_VEL
LIN {X 0,Y 257.944,Z 208.887,A -85,B 0,C 180,E1 -18413.171,E2 -18413.171} C_VEL
LIN {X 0,Y 257.687,Z 212.071,A -85,B 0,C 180,E1 -18416.006,E2 -18416.006} C_VEL
LIN {X 0,Y 256.693,Z 217.281,A -85,B 0,C 180,E1 -18420.473,E2 -18420.473} C_VEL
LIN {X 0,Y 256.56,Z 217.999,A -85,B 0,C 180,E1 -18421.081,E2 -18421.081} C_VEL
LIN {X 0,Y 260.235,Z 232.098,A -85,B 0,C 180,E1 -18422.294,E2 -18422.294} C_VEL
LIN {X 0,Y 262.636,Z 244.287,A -85,B 0,C 180,E1 -18423.55,E2 -18423.55} C_VEL
LIN {X 0,Y 263.981,Z 255.17,A -85,B 0,C 180,E1 -18424.849,E2 -18424.849} C_VEL
LIN {X 0,Y 264.732,Z 267.165,A -85,B 0,C 180,E1 -18426.533,E2 -18426.533} C_VEL
LIN {X 0,Y 264.51,Z 271.079,A -85,B 0,C 180,E1 -18427.133,E2 -18427.133} C_VEL
LIN {X 0,Y 262.414,Z 281.251,A -85,B 0,C 180,E1 -18428.804,E2 -18428.804} C_VEL
LIN {X 0,Y 260.314,Z 291.26,A -85,B 0,C 180,E1 -18430.898,E2 -18430.898} C_VEL
LIN {X 0,Y 258.56,Z 299.353,A -85,B 0,C 180,E1 -18433.01,E2 -18433.01} C_VEL
LIN {X 0,Y 256.963,Z 306.545,A -85,B 0,C 180,E1 -18435.345,E2 -18435.345} C_VEL
LIN {X 0,Y 255.849,Z 311.401,A -85,B 0,C 180,E1 -18437.305,E2 -18437.305} C_VEL
LIN {X 0,Y 254.976,Z 316.127,A -85,B 0,C 180,E1 -18439.679,E2 -18439.679} C_VEL
LIN {X 0,Y 254.373,Z 319.739,A -85,B 0,C 180,E1 -18442.059,E2 -18442.059} C_VEL
LIN {X 0,Y 254.022,Z 322.739,A -85,B 0,C 180,E1 -18444.881,E2 -18444.881} C_VEL
LIN {X 0,Y 253.986,Z 324.003,A -85,B 0,C 180,E1 -18446.827,E2 -18446.827} C_VEL
LIN {X 0,Y 254.015,Z 324.614,A -85,B 0,C 180,E1 -18448.414,E2 -18448.414} C_VEL
LIN {X 0,Y 254.032,Z 324.829,A -85,B 0,C 180,E1 -18450,E2 -18450} C_VEL
LIN {X 0,Y 254.015,Z 324.608,A -85,B 0,C 180,E1 -18451.585,E2 -18451.585} C_VEL
LIN {X 0,Y 253.987,Z 323.993,A -85,B 0,C 180,E1 -18453.172,E2 -18453.172} C_VEL
LIN {X 0,Y 254.022,Z 322.724,A -85,B 0,C 180,E1 -18455.118,E2 -18455.118} C_VEL
LIN {X 0,Y 254.372,Z 319.711,A -85,B 0,C 180,E1 -18457.94,E2 -18457.94} C_VEL
LIN {X 0,Y 254.975,Z 316.084,A -85,B 0,C 180,E1 -18460.321,E2 -18460.321} C_VEL
LIN {X 0,Y 255.847,Z 311.346,A -85,B 0,C 180,E1 -18462.694,E2 -18462.694} C_VEL
LIN {X 0,Y 257.462,Z 304.24,A -85,B 0,C 180,E1 -18465.435,E2 -18465.435} C_VEL
LIN {X 0,Y 259.232,Z 296.528,A -85,B 0,C 180,E1 -18467.758,E2 -18467.758} C_VEL
LIN {X 0,Y 261.217,Z 286.846,A -85,B 0,C 180,E1 -18470.061,E2 -18470.061} C_VEL
LIN {X 0,Y 263.262,Z 276.86,A -85,B 0,C 180,E1 -18471.946,E2 -18471.946} C_VEL
LIN {X 0,Y 264.654,Z 269.621,A -85,B 0,C 180,E1 -18473.059,E2 -18473.059} C_VEL
LIN {X 0,Y 264.314,Z 259.204,A -85,B 0,C 180,E1 -18474.589,E2 -18474.589} C_VEL
LIN {X 0,Y 263.183,Z 247.918,A -85,B 0,C 180,E1 -18476.009,E2 -18476.009} C_VEL
LIN {X 0,Y 261.043,Z 235.797,A -85,B 0,C 180,E1 -18477.32,E2 -18477.32} C_VEL
LIN {X 0,Y 257.869,Z 223.15,A -85,B 0,C 180,E1 -18478.48,E2 -18478.48} C_VEL
LIN {X 0,Y 256.567,Z 218.004,A -85,B 0,C 180,E1 -18478.884,E2 -18478.884} C_VEL
LIN {X 0,Y 257.502,Z 213.089,A -85,B 0,C 180,E1 -18483.083,E2 -18483.083} C_VEL
LIN {X 0,Y 257.904,Z 210.693,A -85,B 0,C 180,E1 -18485.163,E2 -18485.163} C_VEL
LIN {X 0,Y 257.944,Z 206.719,A -85,B 0,C 180,E1 -18488.804,E2 -18488.804} C_VEL
LIN {X 0,Y 257.686,Z 204.569,A -85,B 0,C 180,E1 -18490.886,E2 -18490.886} C_VEL
LIN {X 0,Y 256.867,Z 200.263,A -85,B 0,C 180,E1 -18495.346,E2 -18495.346} C_VEL
LIN {X 0,Y 256.375,Z 197.068,A -85,B 0,C 180,E1 -18498.859,E2 -18498.859} C_VEL
LIN {X 0,Y 256.076,Z 195.586,A -85,B 0,C 180,E1 -18500.859,E2 -18500.859} C_VEL
LIN {X 0,Y 256.078,Z 195.588,A -85,B 0,C 180,E1 -18504.806,E2 -18504.806} C_VEL
LIN {X 0,Y 256.091,Z 195.586,A -85,B 0,C 180,E1 -18508.572,E2 -18508.572} C_VEL
LIN {X 0,Y 256.136,Z 195.581,A -85,B 0,C 180,E1 -18512.196,E2 -18512.196} C_VEL
LIN {X 0,Y 256.141,Z 195.582,A -85,B 0,C 180,E1 -18515.696,E2 -18515.696} C_VEL
LIN {X 0,Y 256.161,Z 195.578,A -85,B 0,C 180,E1 -18519.104,E2 -18519.104} C_VEL
LIN {X 0,Y 256.298,Z 195.559,A -85,B 0,C 180,E1 -18524.085,E2 -18524.085} C_VEL
LIN {X 0,Y 256.293,Z 195.557,A -85,B 0,C 180,E1 -18528.933,E2 -18528.933} C_VEL
LIN {X 0,Y 256.466,Z 195.537,A -85,B 0,C 180,E1 -18532.125,E2 -18532.125} C_VEL
LIN {X 0,Y 256.49,Z 195.537,A -85,B 0,C 180,E1 -18536.859,E2 -18536.859} C_VEL
LIN {X 0,Y 256.764,Z 195.5,A -85,B 0,C 180,E1 -18540,E2 -18540} C_VEL
LIN {X 0,Y 256.49,Z 195.535,A -85,B 0,C 180,E1 -18543.142,E2 -18543.142} C_VEL
LIN {X 0,Y 256.488,Z 195.534,A -85,B 0,C 180,E1 -18547.875,E2 -18547.875} C_VEL
LIN {X 0,Y 256.294,Z 195.559,A -85,B 0,C 180,E1 -18551.067,E2 -18551.067} C_VEL
LIN {X 0,Y 256.299,Z 195.559,A -85,B 0,C 180,E1 -18555.915,E2 -18555.915} C_VEL
LIN {X 0,Y 256.166,Z 195.573,A -85,B 0,C 180,E1 -18560.895,E2 -18560.895} C_VEL
LIN {X 0,Y 256.187,Z 195.572,A -85,B 0,C 180,E1 -18565.139,E2 -18565.139} C_VEL
LIN {X 0,Y 256.11,Z 195.584,A -85,B 0,C 180,E1 -18569.6,E2 -18569.6} C_VEL
LIN {X 0,Y 256.067,Z 195.59,A -85,B 0,C 180,E1 -18573.293,E2 -18573.293} C_VEL
LIN {X 0,Y 256.109,Z 195.583,A -85,B 0,C 180,E1 -18577.27,E2 -18577.27} C_VEL
LIN {X 0,Y 256.054,Z 195.593,A -85,B 0,C 180,E1 -18581.204,E2 -18581.204} C_VEL
LIN {X 0,Y 256.04,Z 195.591,A -85,B 0,C 180,E1 -18585.535,E2 -18585.535} C_VEL
LIN {X 0,Y 256.063,Z 195.591,A -85,B 0,C 180,E1 -18588.799,E2 -18588.799} C_VEL
LIN {X 0,Y 256.254,Z 196.928,A -85,B 0,C 180,E1 -18590.892,E2 -18590.892} C_VEL
LIN {X 0,Y 256.351,Z 198.449,A -85,B 0,C 180,E1 -18592.905,E2 -18592.905} C_VEL
LIN {X 0,Y 256.171,Z 201.531,A -85,B 0,C 180,E1 -18596.723,E2 -18596.723} C_VEL
LIN {X 0,Y 255.862,Z 204.652,A -85,B 0,C 180,E1 -18600.369,E2 -18600.369} C_VEL
LIN {X 0,Y 255.799,Z 205.287,A -85,B 0,C 180,E1 -18601.095,E2 -18601.095} C_VEL
LIN {X 0,Y 256.751,Z 208.398,A -85,B 0,C 180,E1 -18601.375,E2 -18601.375} C_VEL
LIN {X 0,Y 260.796,Z 220.475,A -85,B 0,C 180,E1 -18602.599,E2 -18602.599} C_VEL
LIN {X 0,Y 263.951,Z 232.762,A -85,B 0,C 180,E1 -18604.022,E2 -18604.022} C_VEL
LIN {X 0,Y 265.588,Z 242.371,A -85,B 0,C 180,E1 -18605.279,E2 -18605.279} C_VEL
LIN {X 0,Y 266.447,Z 249.562,A -85,B 0,C 180,E1 -18606.335,E2 -18606.335} C_VEL
LIN {X 0,Y 264.516,Z 260.756,A -85,B 0,C 180,E1 -18607.958,E2 -18607.958} C_VEL
LIN {X 0,Y 262.792,Z 270.062,A -85,B 0,C 180,E1 -18609.656,E2 -18609.656} C_VEL
LIN {X 0,Y 260.981,Z 278.541,A -85,B 0,C 180,E1 -18611.554,E2 -18611.554} C_VEL
LIN {X 0,Y 259.009,Z 286.787,A -85,B 0,C 180,E1 -18613.852,E2 -18613.852} C_VEL
LIN {X 0,Y 257.691,Z 292.423,A -85,B 0,C 180,E1 -18615.792,E2 -18615.792} C_VEL
LIN {X 0,Y 256.359,Z 297.918,A -85,B 0,C 180,E1 -18618.135,E2 -18618.135} C_VEL
LIN {X 0,Y 255.391,Z 302.227,A -85,B 0,C 180,E1 -18620.497,E2 -18620.497} C_VEL
LIN {X 0,Y 254.646,Z 306.181,A -85,B 0,C 180,E1 -18623.501,E2 -18623.501} C_VEL
LIN {X 0,Y 254.373,Z 307.749,A -85,B 0,C 180,E1 -18625.246,E2 -18625.246} C_VEL
LIN {X 0,Y 254.209,Z 308.74,A -85,B 0,C 180,E1 -18626.831,E2 -18626.831} C_VEL
LIN {X 0,Y 254.106,Z 309.349,A -85,B 0,C 180,E1 -18628.416,E2 -18628.416} C_VEL
LIN {X 0,Y 254.066,Z 309.578,A -85,B 0,C 180,E1 -18630,E2 -18630} C_VEL
LIN {X 0,Y 254.105,Z 309.384,A -85,B 0,C 180,E1 -18631.585,E2 -18631.585} C_VEL
LIN {X 0,Y 254.207,Z 308.798,A -85,B 0,C 180,E1 -18633.17,E2 -18633.17} C_VEL
LIN {X 0,Y 254.606,Z 306.475,A -85,B 0,C 180,E1 -18636.34,E2 -18636.34} C_VEL
LIN {X 0,Y 255.156,Z 303.609,A -85,B 0,C 180,E1 -18638.714,E2 -18638.714} C_VEL
LIN {X 0,Y 255.963,Z 299.722,A -85,B 0,C 180,E1 -18641.082,E2 -18641.082} C_VEL
LIN {X 0,Y 257.146,Z 294.703,A -85,B 0,C 180,E1 -18643.434,E2 -18643.434} C_VEL
LIN {X 0,Y 258.622,Z 288.382,A -85,B 0,C 180,E1 -18645.769,E2 -18645.769} C_VEL
LIN {X 0,Y 260.596,Z 280.466,A -85,B 0,C 180,E1 -18648.068,E2 -18648.068} C_VEL
LIN {X 0,Y 262.437,Z 272.397,A -85,B 0,C 180,E1 -18649.965,E2 -18649.965} C_VEL
LIN {X 0,Y 264.222,Z 262.557,A -85,B 0,C 180,E1 -18651.863,E2 -18651.863} C_VEL
LIN {X 0,Y 266.251,Z 251.597,A -85,B 0,C 180,E1 -18653.512,E2 -18653.512} C_VEL
LIN {X 0,Y 266.32,Z 247.72,A -85,B 0,C 180,E1 -18654.069,E2 -18654.069} C_VEL
LIN {X 0,Y 264.805,Z 237.302,A -85,B 0,C 180,E1 -18655.528,E2 -18655.528} C_VEL
LIN {X 0,Y 262.193,Z 225.501,A -85,B 0,C 180,E1 -18656.97,E2 -18656.97} C_VEL
LIN {X 0,Y 258.6,Z 213.576,A -85,B 0,C 180,E1 -18658.25,E2 -18658.25} C_VEL
LIN {X 0,Y 255.891,Z 205.823,A -85,B 0,C 180,E1 -18658.988,E2 -18658.988} C_VEL
LIN {X 0,Y 255.798,Z 205.287,A -85,B 0,C 180,E1 -18659.042,E2 -18659.042} C_VEL
LIN {X 0,Y 256.072,Z 202.982,A -85,B 0,C 180,E1 -18661.7,E2 -18661.7} C_VEL
LIN {X 0,Y 256.304,Z 200.102,A -85,B 0,C 180,E1 -18665.158,E2 -18665.158} C_VEL
LIN {X 0,Y 256.357,Z 198.38,A -85,B 0,C 180,E1 -18667.341,E2 -18667.341} C_VEL
LIN {X 0,Y 256.027,Z 195.591,A -85,B 0,C 180,E1 -18671.209,E2 -18671.209} C_VEL
LIN {X 0,Y 256.041,Z 195.591,A -85,B 0,C 180,E1 -18675.534,E2 -18675.534} C_VEL
LIN {X 0,Y 256.056,Z 195.591,A -85,B 0,C 180,E1 -18678.797,E2 -18678.797} C_VEL
LIN {X 0,Y 256.128,Z 195.581,A -85,B 0,C 180,E1 -18682.867,E2 -18682.867} C_VEL
LIN {X 0,Y 256.069,Z 195.589,A -85,B 0,C 180,E1 -18686.707,E2 -18686.707} C_VEL
LIN {X 0,Y 256.105,Z 195.583,A -85,B 0,C 180,E1 -18690.399,E2 -18690.399} C_VEL
LIN {X 0,Y 256.19,Z 195.572,A -85,B 0,C 180,E1 -18694.862,E2 -18694.862} C_VEL
LIN {X 0,Y 256.169,Z 195.574,A -85,B 0,C 180,E1 -18699.105,E2 -18699.105} C_VEL
LIN {X 0,Y 256.302,Z 195.56,A -85,B 0,C 180,E1 -18704.085,E2 -18704.085} C_VEL
LIN {X 0,Y 256.297,Z 195.558,A -85,B 0,C 180,E1 -18708.933,E2 -18708.933} C_VEL
LIN {X 0,Y 256.491,Z 195.534,A -85,B 0,C 180,E1 -18712.125,E2 -18712.125} C_VEL
LIN {X 0,Y 256.492,Z 195.535,A -85,B 0,C 180,E1 -18716.858,E2 -18716.858} C_VEL
LIN {X 0,Y 256.767,Z 195.499,A -85,B 0,C 180,E1 -18720,E2 -18720} C_VEL
LIN {X 0,Y 256.493,Z 195.537,A -85,B 0,C 180,E1 -18723.141,E2 -18723.141} C_VEL
LIN {X 0,Y 256.47,Z 195.537,A -85,B 0,C 180,E1 -18727.875,E2 -18727.875} C_VEL
LIN {X 0,Y 256.299,Z 195.561,A -85,B 0,C 180,E1 -18731.066,E2 -18731.066} C_VEL
LIN {X 0,Y 256.258,Z 195.567,A -85,B 0,C 180,E1 -18734.29,E2 -18734.29} C_VEL
LIN {X 0,Y 256.211,Z 195.57,A -85,B 0,C 180,E1 -18737.562,E2 -18737.562} C_VEL
LIN {X 0,Y 256.155,Z 195.577,A -85,B 0,C 180,E1 -18741.117,E2 -18741.117} C_VEL
LIN {X 0,Y 256.172,Z 195.574,A -85,B 0,C 180,E1 -18745.13,E2 -18745.13} C_VEL
LIN {X 0,Y 256.104,Z 195.585,A -85,B 0,C 180,E1 -18749.522,E2 -18749.522} C_VEL
LIN {X 0,Y 255.455,Z 195.672,A -85,B 0,C 180,E1 -18750.834,E2 -18750.834} C_VEL
LIN {X 0,Y 252.612,Z 196.032,A -85,B 0,C 180,E1 -18752.972,E2 -18752.972} C_VEL
LIN {X 0,Y 250.177,Z 196.332,A -85,B 0,C 180,E1 -18754.713,E2 -18754.713} C_VEL
LIN {X 0,Y 249.116,Z 196.458,A -85,B 0,C 180,E1 -18756.062,E2 -18756.062} C_VEL
LIN {X 0,Y 249.021,Z 196.468,A -85,B 0,C 180,E1 -18756.52,E2 -18756.52} C_VEL
LIN {X 0,Y 249.068,Z 196.645,A -85,B 0,C 180,E1 -18758.89,E2 -18758.89} C_VEL
LIN {X 0,Y 249.635,Z 200.069,A -85,B 0,C 180,E1 -18762.947,E2 -18762.947} C_VEL
LIN {X 0,Y 250.422,Z 204.382,A -85,B 0,C 180,E1 -18767.658,E2 -18767.658} C_VEL
LIN {X 0,Y 250.799,Z 206.535,A -85,B 0,C 180,E1 -18769.87,E2 -18769.87} C_VEL
LIN {X 0,Y 250.927,Z 209.729,A -85,B 0,C 180,E1 -18772.974,E2 -18772.974} C_VEL
LIN {X 0,Y 250.676,Z 212.907,A -85,B 0,C 180,E1 -18775.894,E2 -18775.894} C_VEL
LIN {X 0,Y 249.684,Z 217.8,A -85,B 0,C 180,E1 -18780.214,E2 -18780.214} C_VEL
LIN {X 0,Y 253.282,Z 231.346,A -85,B 0,C 180,E1 -18781.426,E2 -18781.426} C_VEL
LIN {X 0,Y 255.543,Z 242.146,A -85,B 0,C 180,E1 -18782.57,E2 -18782.57} C_VEL
LIN {X 0,Y 257.23,Z 254.433,A -85,B 0,C 180,E1 -18784.078,E2 -18784.078} C_VEL
LIN {X 0,Y 257.915,Z 265.04,A -85,B 0,C 180,E1 -18785.589,E2 -18785.589} C_VEL
LIN {X 0,Y 257.959,Z 270.869,A -85,B 0,C 180,E1 -18786.518,E2 -18786.518} C_VEL
LIN {X 0,Y 255.783,Z 281.041,A -85,B 0,C 180,E1 -18788.227,E2 -18788.227} C_VEL
LIN {X 0,Y 253.743,Z 290.37,A -85,B 0,C 180,E1 -18790.208,E2 -18790.208} C_VEL
LIN {X 0,Y 252.102,Z 297.782,A -85,B 0,C 180,E1 -18792.142,E2 -18792.142} C_VEL
LIN {X 0,Y 250.314,Z 305.216,A -85,B 0,C 180,E1 -18794.53,E2 -18794.53} C_VEL
LIN {X 0,Y 248.886,Z 311.188,A -85,B 0,C 180,E1 -18796.944,E2 -18796.944} C_VEL
LIN {X 0,Y 247.951,Z 315.914,A -85,B 0,C 180,E1 -18799.383,E2 -18799.383} C_VEL
LIN {X 0,Y 247.34,Z 319.527,A -85,B 0,C 180,E1 -18801.832,E2 -18801.832} C_VEL
LIN {X 0,Y 247.075,Z 321.391,A -85,B 0,C 180,E1 -18803.466,E2 -18803.466} C_VEL
LIN {X 0,Y 246.922,Z 322.79,A -85,B 0,C 180,E1 -18805.101,E2 -18805.101} C_VEL
LIN {X 0,Y 246.889,Z 323.79,A -85,B 0,C 180,E1 -18806.736,E2 -18806.736} C_VEL
LIN {X 0,Y 246.924,Z 324.402,A -85,B 0,C 180,E1 -18808.369,E2 -18808.369} C_VEL
LIN {X 0,Y 246.962,Z 324.617,A -85,B 0,C 180,E1 -18810,E2 -18810} C_VEL
LIN {X 0,Y 246.924,Z 324.395,A -85,B 0,C 180,E1 -18811.631,E2 -18811.631} C_VEL
LIN {X 0,Y 246.889,Z 323.78,A -85,B 0,C 180,E1 -18813.263,E2 -18813.263} C_VEL
LIN {X 0,Y 246.944,Z 322.661,A -85,B 0,C 180,E1 -18815.063,E2 -18815.063} C_VEL
LIN {X 0,Y 247.074,Z 321.37,A -85,B 0,C 180,E1 -18816.533,E2 -18816.533} C_VEL
LIN {X 0,Y 247.518,Z 318.421,A -85,B 0,C 180,E1 -18818.984,E2 -18818.984} C_VEL
LIN {X 0,Y 248.237,Z 314.433,A -85,B 0,C 180,E1 -18821.43,E2 -18821.43} C_VEL
LIN {X 0,Y 249.535,Z 308.306,A -85,B 0,C 180,E1 -18824.266,E2 -18824.266} C_VEL
LIN {X 0,Y 251.202,Z 301.622,A -85,B 0,C 180,E1 -18826.664,E2 -18826.664} C_VEL
LIN {X 0,Y 253.23,Z 292.955,A -85,B 0,C 180,E1 -18829.136,E2 -18829.136} C_VEL
LIN {X 0,Y 254.92,Z 284.824,A -85,B 0,C 180,E1 -18831.002,E2 -18831.002} C_VEL
LIN {X 0,Y 257.183,Z 274.324,A -85,B 0,C 180,E1 -18832.917,E2 -18832.917} C_VEL
LIN {X 0,Y 257.941,Z 269.398,A -85,B 0,C 180,E1 -18833.696,E2 -18833.696} C_VEL
LIN {X 0,Y 257.564,Z 258.976,A -85,B 0,C 180,E1 -18835.278,E2 -18835.278} C_VEL
LIN {X 0,Y 256.335,Z 247.091,A -85,B 0,C 180,E1 -18836.824,E2 -18836.824} C_VEL
LIN {X 0,Y 254.117,Z 234.905,A -85,B 0,C 180,E1 -18838.178,E2 -18838.178} C_VEL
LIN {X 0,Y 250.707,Z 221.728,A -85,B 0,C 180,E1 -18839.431,E2 -18839.431} C_VEL
LIN {X 0,Y 249.681,Z 217.781,A -85,B 0,C 180,E1 -18839.771,E2 -18839.771} C_VEL
LIN {X 0,Y 250.675,Z 212.868,A -85,B 0,C 180,E1 -18844.105,E2 -18844.105} C_VEL
LIN {X 0,Y 250.952,Z 209.694,A -85,B 0,C 180,E1 -18847.021,E2 -18847.021} C_VEL
LIN {X 0,Y 250.809,Z 206.495,A -85,B 0,C 180,E1 -18850.127,E2 -18850.127} C_VEL
LIN {X 0,Y 250.281,Z 203.616,A -85,B 0,C 180,E1 -18853.106,E2 -18853.106} C_VEL
LIN {X 0,Y 249.559,Z 199.654,A -85,B 0,C 180,E1 -18857.477,E2 -18857.477} C_VEL
LIN {X 0,Y 249.02,Z 196.468,A -85,B 0,C 180,E1 -18861.36,E2 -18861.36} C_VEL
LIN {X 0,Y 249.042,Z 196.464,A -85,B 0,C 180,E1 -18865.639,E2 -18865.639} C_VEL
LIN {X 0,Y 249.046,Z 196.463,A -85,B 0,C 180,E1 -18869.472,E2 -18869.472} C_VEL
LIN {X 0,Y 249.067,Z 196.461,A -85,B 0,C 180,E1 -18873.161,E2 -18873.161} C_VEL
LIN {X 0,Y 249.06,Z 196.462,A -85,B 0,C 180,E1 -18876.731,E2 -18876.731} C_VEL
LIN {X 0,Y 249.108,Z 196.456,A -85,B 0,C 180,E1 -18880.211,E2 -18880.211} C_VEL
LIN {X 0,Y 249.24,Z 196.44,A -85,B 0,C 180,E1 -18883.622,E2 -18883.622} C_VEL
LIN {X 0,Y 249.241,Z 196.436,A -85,B 0,C 180,E1 -18888.616,E2 -18888.616} C_VEL
LIN {X 0,Y 249.416,Z 196.416,A -85,B 0,C 180,E1 -18891.901,E2 -18891.901} C_VEL
LIN {X 0,Y 249.28,Z 196.434,A -85,B 0,C 180,E1 -18895.148,E2 -18895.148} C_VEL
LIN {X 0,Y 249.673,Z 196.383,A -85,B 0,C 180,E1 -18898.387,E2 -18898.387} C_VEL
LIN {X 0,Y 249.672,Z 196.383,A -85,B 0,C 180,E1 -18901.613,E2 -18901.613} C_VEL
LIN {X 0,Y 249.421,Z 196.415,A -85,B 0,C 180,E1 -18906.628,E2 -18906.628} C_VEL
LIN {X 0,Y 249.341,Z 196.424,A -85,B 0,C 180,E1 -18909.737,E2 -18909.737} C_VEL
LIN {X 0,Y 249.204,Z 196.442,A -85,B 0,C 180,E1 -18914.704,E2 -18914.704} C_VEL
LIN {X 0,Y 249.138,Z 196.452,A -85,B 0,C 180,E1 -18918.078,E2 -18918.078} C_VEL
LIN {X 0,Y 249.086,Z 196.456,A -85,B 0,C 180,E1 -18921.518,E2 -18921.518} C_VEL
LIN {X 0,Y 249.129,Z 196.453,A -85,B 0,C 180,E1 -18925.482,E2 -18925.482} C_VEL
LIN {X 0,Y 249.079,Z 196.458,A -85,B 0,C 180,E1 -18928.993,E2 -18928.993} C_VEL
LIN {X 0,Y 249.03,Z 196.464,A -85,B 0,C 180,E1 -18932.426,E2 -18932.426} C_VEL
LIN {X 0,Y 249.025,Z 196.465,A -85,B 0,C 180,E1 -18936.346,E2 -18936.346} C_VEL
LIN {X 0,Y 249.005,Z 196.468,A -85,B 0,C 180,E1 -18940.479,E2 -18940.479} C_VEL
LIN {X 0,Y 248.985,Z 196.472,A -85,B 0,C 180,E1 -18944.884,E2 -18944.884} C_VEL
LIN {X 0,Y 249.009,Z 196.469,A -85,B 0,C 180,E1 -18947.362,E2 -18947.362} C_VEL
LIN {X 0,Y 249.128,Z 197.201,A -85,B 0,C 180,E1 -18949.613,E2 -18949.613} C_VEL
LIN {X 0,Y 249.296,Z 199.019,A -85,B 0,C 180,E1 -18952.126,E2 -18952.126} C_VEL
LIN {X 0,Y 249.216,Z 201.755,A -85,B 0,C 180,E1 -18955.667,E2 -18955.667} C_VEL
LIN {X 0,Y 248.878,Z 205.275,A -85,B 0,C 180,E1 -18959.914,E2 -18959.914} C_VEL
LIN {X 0,Y 248.843,Z 205.528,A -85,B 0,C 180,E1 -18960.209,E2 -18960.209} C_VEL
LIN {X 0,Y 249.877,Z 208.683,A -85,B 0,C 180,E1 -18960.513,E2 -18960.513} C_VEL
LIN {X 0,Y 254.144,Z 221.321,A -85,B 0,C 180,E1 -18961.864,E2 -18961.864} C_VEL
LIN {X 0,Y 257.133,Z 232.892,A -85,B 0,C 180,E1 -18963.268,E2 -18963.268} C_VEL
LIN {X 0,Y 258.971,Z 243.525,A -85,B 0,C 180,E1 -18964.723,E2 -18964.723} C_VEL
LIN {X 0,Y 259.79,Z 251.115,A -85,B 0,C 180,E1 -18965.889,E2 -18965.889} C_VEL
LIN {X 0,Y 257.721,Z 262.127,A -85,B 0,C 180,E1 -18967.557,E2 -18967.557} C_VEL
LIN {X 0,Y 255.801,Z 272.081,A -85,B 0,C 180,E1 -18969.495,E2 -18969.495} C_VEL
LIN {X 0,Y 253.558,Z 281.714,A -85,B 0,C 180,E1 -18971.831,E2 -18971.831} C_VEL
LIN {X 0,Y 251.592,Z 289.394,A -85,B 0,C 180,E1 -18974.196,E2 -18974.196} C_VEL
LIN {X 0,Y 249.847,Z 296.441,A -85,B 0,C 180,E1 -18976.996,E2 -18976.996} C_VEL
LIN {X 0,Y 248.673,Z 301.134,A -85,B 0,C 180,E1 -18979.415,E2 -18979.415} C_VEL
LIN {X 0,Y 247.925,Z 304.719,A -85,B 0,C 180,E1 -18981.852,E2 -18981.852} C_VEL
LIN {X 0,Y 247.523,Z 306.691,A -85,B 0,C 180,E1 -18983.602,E2 -18983.602} C_VEL
LIN {X 0,Y 247.13,Z 308.953,A -85,B 0,C 180,E1 -18986.74,E2 -18986.74} C_VEL
LIN {X 0,Y 247.038,Z 309.561,A -85,B 0,C 180,E1 -18988.37,E2 -18988.37} C_VEL
LIN {X 0,Y 246.996,Z 309.79,A -85,B 0,C 180,E1 -18990,E2 -18990} C_VEL
LIN {X 0,Y 247.038,Z 309.596,A -85,B 0,C 180,E1 -18991.631,E2 -18991.631} C_VEL
LIN {X 0,Y 247.128,Z 309.011,A -85,B 0,C 180,E1 -18993.261,E2 -18993.261} C_VEL
LIN {X 0,Y 247.547,Z 306.688,A -85,B 0,C 180,E1 -18996.521,E2 -18996.521} C_VEL
LIN {X 0,Y 248.123,Z 303.822,A -85,B 0,C 180,E1 -18998.963,E2 -18998.963} C_VEL
LIN {X 0,Y 249.007,Z 299.933,A -85,B 0,C 180,E1 -19001.395,E2 -19001.395} C_VEL
LIN {X 0,Y 250.232,Z 294.915,A -85,B 0,C 180,E1 -19003.812,E2 -19003.812} C_VEL
LIN {X 0,Y 251.797,Z 288.593,A -85,B 0,C 180,E1 -19006.208,E2 -19006.208} C_VEL
LIN {X 0,Y 253.844,Z 280.677,A -85,B 0,C 180,E1 -19008.566,E2 -19008.566} C_VEL
LIN {X 0,Y 255.762,Z 272.607,A -85,B 0,C 180,E1 -19010.509,E2 -19010.509} C_VEL
LIN {X 0,Y 257.412,Z 263.833,A -85,B 0,C 180,E1 -19012.261,E2 -19012.261} C_VEL
LIN {X 0,Y 259.549,Z 253.069,A -85,B 0,C 180,E1 -19013.964,E2 -19013.964} C_VEL
LIN {X 0,Y 259.744,Z 249.513,A -85,B 0,C 180,E1 -19014.483,E2 -19014.483} C_VEL
LIN {X 0,Y 258.421,Z 239.811,A -85,B 0,C 180,E1 -19015.929,E2 -19015.929} C_VEL
LIN {X 0,Y 256.201,Z 228.879,A -85,B 0,C 180,E1 -19017.366,E2 -19017.366} C_VEL
LIN {X 0,Y 252.753,Z 216.866,A -85,B 0,C 180,E1 -19018.77,E2 -19018.77} C_VEL
LIN {X 0,Y 248.903,Z 205.868,A -85,B 0,C 180,E1 -19019.891,E2 -19019.891} C_VEL
LIN {X 0,Y 248.873,Z 205.484,A -85,B 0,C 180,E1 -19019.976,E2 -19019.976} C_VEL
LIN {X 0,Y 249.231,Z 201.868,A -85,B 0,C 180,E1 -19024.332,E2 -19024.332} C_VEL
LIN {X 0,Y 249.299,Z 199.143,A -85,B 0,C 180,E1 -19027.875,E2 -19027.875} C_VEL
LIN {X 0,Y 249.116,Z 197.263,A -85,B 0,C 180,E1 -19030.457,E2 -19030.457} C_VEL
LIN {X 0,Y 248.977,Z 196.469,A -85,B 0,C 180,E1 -19032.784,E2 -19032.784} C_VEL
LIN {X 0,Y 249.011,Z 196.468,A -85,B 0,C 180,E1 -19037.361,E2 -19037.361} C_VEL
LIN {X 0,Y 249.026,Z 196.465,A -85,B 0,C 180,E1 -19041.619,E2 -19041.619} C_VEL
LIN {X 0,Y 249.045,Z 196.461,A -85,B 0,C 180,E1 -19045.639,E2 -19045.639} C_VEL
LIN {X 0,Y 249.049,Z 196.461,A -85,B 0,C 180,E1 -19049.473,E2 -19049.473} C_VEL
LIN {X 0,Y 249.074,Z 196.457,A -85,B 0,C 180,E1 -19053.162,E2 -19053.162} C_VEL
LIN {X 0,Y 249.081,Z 196.456,A -85,B 0,C 180,E1 -19056.733,E2 -19056.733} C_VEL
LIN {X 0,Y 249.113,Z 196.455,A -85,B 0,C 180,E1 -19060.212,E2 -19060.212} C_VEL
LIN {X 0,Y 249.244,Z 196.437,A -85,B 0,C 180,E1 -19063.622,E2 -19063.622} C_VEL
LIN {X 0,Y 249.245,Z 196.437,A -85,B 0,C 180,E1 -19068.616,E2 -19068.616} C_VEL
LIN {X 0,Y 249.436,Z 196.414,A -85,B 0,C 180,E1 -19071.901,E2 -19071.901} C_VEL
LIN {X 0,Y 249.428,Z 196.415,A -85,B 0,C 180,E1 -19076.769,E2 -19076.769} C_VEL
LIN {X 0,Y 249.73,Z 196.375,A -85,B 0,C 180,E1 -19080,E2 -19080} C_VEL
LIN {X 0,Y 249.429,Z 196.417,A -85,B 0,C 180,E1 -19083.23,E2 -19083.23} C_VEL
LIN {X 0,Y 249.43,Z 196.416,A -85,B 0,C 180,E1 -19086.471,E2 -19086.471} C_VEL
LIN {X 0,Y 249.345,Z 196.425,A -85,B 0,C 180,E1 -19089.736,E2 -19089.736} C_VEL
LIN {X 0,Y 249.208,Z 196.445,A -85,B 0,C 180,E1 -19094.703,E2 -19094.703} C_VEL
LIN {X 0,Y 249.14,Z 196.453,A -85,B 0,C 180,E1 -19098.077,E2 -19098.077} C_VEL
LIN {X 0,Y 249.086,Z 196.458,A -85,B 0,C 180,E1 -19101.518,E2 -19101.518} C_VEL
LIN {X 0,Y 249.119,Z 196.454,A -85,B 0,C 180,E1 -19105.475,E2 -19105.475} C_VEL
LIN {X 0,Y 249.046,Z 196.461,A -85,B 0,C 180,E1 -19109.509,E2 -19109.509} C_VEL
LIN {X 0,Y 249.032,Z 196.468,A -85,B 0,C 180,E1 -19112.426,E2 -19112.426} C_VEL
LIN {X 0,Y 249.021,Z 196.468,A -85,B 0,C 180,E1 -19116.52,E2 -19116.52} C_VEL
LIN {X 0,Y 248.376,Z 196.805,A -85,B 0,C 180,E1 -19117.868,E2 -19117.868} C_VEL
LIN {X 0,Y 246.914,Z 197.669,A -85,B 0,C 180,E1 -19119.185,E2 -19119.185} C_VEL
LIN {X 0,Y 243.601,Z 200.236,A -85,B 0,C 180,E1 -19121.816,E2 -19121.816} C_VEL
LIN {X 0,Y 242.781,Z 201.589,A -85,B 0,C 180,E1 -19123.177,E2 -19123.177} C_VEL
LIN {X 0,Y 242.767,Z 202.004,A -85,B 0,C 180,E1 -19123.638,E2 -19123.638} C_VEL
LIN {X 0,Y 243.593,Z 206.472,A -85,B 0,C 180,E1 -19128.602,E2 -19128.602} C_VEL
LIN {X 0,Y 243.843,Z 208.887,A -85,B 0,C 180,E1 -19131.095,E2 -19131.095} C_VEL
LIN {X 0,Y 243.841,Z 211.655,A -85,B 0,C 180,E1 -19133.806,E2 -19133.806} C_VEL
LIN {X 0,Y 243.383,Z 214.914,A -85,B 0,C 180,E1 -19136.868,E2 -19136.868} C_VEL
LIN {X 0,Y 242.833,Z 217.553,A -85,B 0,C 180,E1 -19139.269,E2 -19139.269} C_VEL
LIN {X 0,Y 244.455,Z 223.496,A -85,B 0,C 180,E1 -19139.805,E2 -19139.805} C_VEL
LIN {X 0,Y 247.553,Z 235.65,A -85,B 0,C 180,E1 -19141.045,E2 -19141.045} C_VEL
LIN {X 0,Y 249.757,Z 247.913,A -85,B 0,C 180,E1 -19142.496,E2 -19142.496} C_VEL
LIN {X 0,Y 250.925,Z 259.855,A -85,B 0,C 180,E1 -19144.127,E2 -19144.127} C_VEL
LIN {X 0,Y 251.28,Z 270.655,A -85,B 0,C 180,E1 -19145.855,E2 -19145.855} C_VEL
LIN {X 0,Y 249.198,Z 280.83,A -85,B 0,C 180,E1 -19147.621,E2 -19147.621} C_VEL
LIN {X 0,Y 247.074,Z 289.993,A -85,B 0,C 180,E1 -19149.607,E2 -19149.607} C_VEL
LIN {X 0,Y 245.345,Z 297.57,A -85,B 0,C 180,E1 -19151.633,E2 -19151.633} C_VEL
LIN {X 0,Y 243.459,Z 305.004,A -85,B 0,C 180,E1 -19154.083,E2 -19154.083} C_VEL
LIN {X 0,Y 241.936,Z 310.975,A -85,B 0,C 180,E1 -19156.562,E2 -19156.562} C_VEL
LIN {X 0,Y 240.943,Z 315.701,A -85,B 0,C 180,E1 -19159.07,E2 -19159.07} C_VEL
LIN {X 0,Y 240.28,Z 319.313,A -85,B 0,C 180,E1 -19161.59,E2 -19161.59} C_VEL
LIN {X 0,Y 240,Z 321.178,A -85,B 0,C 180,E1 -19163.273,E2 -19163.273} C_VEL
LIN {X 0,Y 239.837,Z 322.659,A -85,B 0,C 180,E1 -19165.078,E2 -19165.078} C_VEL
LIN {X 0,Y 239.835,Z 324.189,A -85,B 0,C 180,E1 -19168.32,E2 -19168.32} C_VEL
LIN {X 0,Y 239.872,Z 324.404,A -85,B 0,C 180,E1 -19170,E2 -19170} C_VEL
LIN {X 0,Y 239.835,Z 324.182,A -85,B 0,C 180,E1 -19171.679,E2 -19171.679} C_VEL
LIN {X 0,Y 239.837,Z 322.644,A -85,B 0,C 180,E1 -19174.921,E2 -19174.921} C_VEL
LIN {X 0,Y 239.999,Z 321.155,A -85,B 0,C 180,E1 -19176.726,E2 -19176.726} C_VEL
LIN {X 0,Y 240.469,Z 318.206,A -85,B 0,C 180,E1 -19179.25,E2 -19179.25} C_VEL
LIN {X 0,Y 241.255,Z 314.218,A -85,B 0,C 180,E1 -19181.766,E2 -19181.766} C_VEL
LIN {X 0,Y 242.647,Z 308.091,A -85,B 0,C 180,E1 -19184.68,E2 -19184.68} C_VEL
LIN {X 0,Y 244.363,Z 301.405,A -85,B 0,C 180,E1 -19187.145,E2 -19187.145} C_VEL
LIN {X 0,Y 246.354,Z 293.371,A -85,B 0,C 180,E1 -19189.509,E2 -19189.509} C_VEL
LIN {X 0,Y 248.268,Z 284.606,A -85,B 0,C 180,E1 -19191.592,E2 -19191.592} C_VEL
LIN {X 0,Y 250.653,Z 274.107,A -85,B 0,C 180,E1 -19193.55,E2 -19193.55} C_VEL
LIN {X 0,Y 251.231,Z 270.476,A -85,B 0,C 180,E1 -19194.149,E2 -19194.149} C_VEL
LIN {X 0,Y 250.92,Z 259.821,A -85,B 0,C 180,E1 -19195.847,E2 -19195.847} C_VEL
LIN {X 0,Y 249.741,Z 247.833,A -85,B 0,C 180,E1 -19197.481,E2 -19197.481} C_VEL
LIN {X 0,Y 247.681,Z 236.379,A -85,B 0,C 180,E1 -19198.84,E2 -19198.84} C_VEL
LIN {X 0,Y 244.549,Z 223.787,A -85,B 0,C 180,E1 -19200.129,E2 -19200.129} C_VEL
LIN {X 0,Y 242.801,Z 217.55,A -85,B 0,C 180,E1 -19200.702,E2 -19200.702} C_VEL
LIN {X 0,Y 243.64,Z 213.688,A -85,B 0,C 180,E1 -19204.228,E2 -19204.228} C_VEL
LIN {X 0,Y 243.941,Z 210.529,A -85,B 0,C 180,E1 -19207.229,E2 -19207.229} C_VEL
LIN {X 0,Y 243.857,Z 208.404,A -85,B 0,C 180,E1 -19209.348,E2 -19209.348} C_VEL
LIN {X 0,Y 243.557,Z 206.262,A -85,B 0,C 180,E1 -19211.58,E2 -19211.58} C_VEL
LIN {X 0,Y 242.762,Z 201.956,A -85,B 0,C 180,E1 -19216.364,E2 -19216.364} C_VEL
LIN {X 0,Y 242.216,Z 198.652,A -85,B 0,C 180,E1 -19220.332,E2 -19220.332} C_VEL
LIN {X 0,Y 242.001,Z 197.341,A -85,B 0,C 180,E1 -19222.02,E2 -19222.02} C_VEL
LIN {X 0,Y 241.979,Z 197.344,A -85,B 0,C 180,E1 -19226.507,E2 -19226.507} C_VEL
LIN {X 0,Y 242.012,Z 197.339,A -85,B 0,C 180,E1 -19230.597,E2 -19230.597} C_VEL
LIN {X 0,Y 242.066,Z 197.334,A -85,B 0,C 180,E1 -19234.183,E2 -19234.183} C_VEL
LIN {X 0,Y 242.025,Z 197.339,A -85,B 0,C 180,E1 -19238.313,E2 -19238.313} C_VEL
LIN {X 0,Y 242.162,Z 197.322,A -85,B 0,C 180,E1 -19243.278,E2 -19243.278} C_VEL
LIN {X 0,Y 242.178,Z 197.315,A -85,B 0,C 180,E1 -19248.279,E2 -19248.279} C_VEL
LIN {X 0,Y 242.37,Z 197.294,A -85,B 0,C 180,E1 -19251.664,E2 -19251.664} C_VEL
LIN {X 0,Y 242.24,Z 197.311,A -85,B 0,C 180,E1 -19255.007,E2 -19255.007} C_VEL
LIN {X 0,Y 242.633,Z 197.26,A -85,B 0,C 180,E1 -19258.34,E2 -19258.34} C_VEL
LIN {X 0,Y 242.633,Z 197.26,A -85,B 0,C 180,E1 -19261.66,E2 -19261.66} C_VEL
LIN {X 0,Y 242.401,Z 197.29,A -85,B 0,C 180,E1 -19266.66,E2 -19266.66} C_VEL
LIN {X 0,Y 242.266,Z 197.306,A -85,B 0,C 180,E1 -19270.024,E2 -19270.024} C_VEL
LIN {X 0,Y 242.165,Z 197.318,A -85,B 0,C 180,E1 -19275.141,E2 -19275.141} C_VEL
LIN {X 0,Y 242.072,Z 197.331,A -85,B 0,C 180,E1 -19278.624,E2 -19278.624} C_VEL
LIN {X 0,Y 242.012,Z 197.34,A -85,B 0,C 180,E1 -19282.18,E2 -19282.18} C_VEL
LIN {X 0,Y 242.065,Z 197.333,A -85,B 0,C 180,E1 -19285.838,E2 -19285.838} C_VEL
LIN {X 0,Y 242.028,Z 197.338,A -85,B 0,C 180,E1 -19289.581,E2 -19289.581} C_VEL
LIN {X 0,Y 241.979,Z 197.344,A -85,B 0,C 180,E1 -19293.493,E2 -19293.493} C_VEL
LIN {X 0,Y 241.983,Z 197.343,A -85,B 0,C 180,E1 -19297.583,E2 -19297.583} C_VEL
LIN {X 0,Y 241.933,Z 197.349,A -85,B 0,C 180,E1 -19301.924,E2 -19301.924} C_VEL
LIN {X 0,Y 241.925,Z 197.352,A -85,B 0,C 180,E1 -19306.574,E2 -19306.574} C_VEL
LIN {X 0,Y 241.963,Z 197.389,A -85,B 0,C 180,E1 -19308.084,E2 -19308.084} C_VEL
LIN {X 0,Y 242.283,Z 200.44,A -85,B 0,C 180,E1 -19312.472,E2 -19312.472} C_VEL
LIN {X 0,Y 242.264,Z 201.982,A -85,B 0,C 180,E1 -19314.536,E2 -19314.536} C_VEL
LIN {X 0,Y 241.898,Z 205.579,A -85,B 0,C 180,E1 -19319.06,E2 -19319.06} C_VEL
LIN {X 0,Y 241.895,Z 205.778,A -85,B 0,C 180,E1 -19319.275,E2 -19319.275} C_VEL
LIN {X 0,Y 242.965,Z 208.988,A -85,B 0,C 180,E1 -19319.589,E2 -19319.589} C_VEL
LIN {X 0,Y 247.185,Z 221.119,A -85,B 0,C 180,E1 -19320.963,E2 -19320.963} C_VEL
LIN {X 0,Y 250.328,Z 233.13,A -85,B 0,C 180,E1 -19322.481,E2 -19322.481} C_VEL
LIN {X 0,Y 252.279,Z 243.754,A -85,B 0,C 180,E1 -19324.003,E2 -19324.003} C_VEL
LIN {X 0,Y 253.129,Z 252.477,A -85,B 0,C 180,E1 -19325.389,E2 -19325.389} C_VEL
LIN {X 0,Y 250.903,Z 263.523,A -85,B 0,C 180,E1 -19327.152,E2 -19327.152} C_VEL
LIN {X 0,Y 249.146,Z 272.297,A -85,B 0,C 180,E1 -19328.921,E2 -19328.921} C_VEL
LIN {X 0,Y 247.16,Z 280.452,A -85,B 0,C 180,E1 -19330.914,E2 -19330.914} C_VEL
LIN {X 0,Y 245.033,Z 288.444,A -85,B 0,C 180,E1 -19333.333,E2 -19333.333} C_VEL
LIN {X 0,Y 243.399,Z 294.851,A -85,B 0,C 180,E1 -19335.793,E2 -19335.793} C_VEL
LIN {X 0,Y 242.056,Z 299.933,A -85,B 0,C 180,E1 -19338.274,E2 -19338.274} C_VEL
LIN {X 0,Y 241.127,Z 303.875,A -85,B 0,C 180,E1 -19340.776,E2 -19340.776} C_VEL
LIN {X 0,Y 240.4,Z 307.162,A -85,B 0,C 180,E1 -19343.711,E2 -19343.711} C_VEL
LIN {X 0,Y 240.054,Z 309.166,A -85,B 0,C 180,E1 -19346.644,E2 -19346.644} C_VEL
LIN {X 0,Y 239.927,Z 310.003,A -85,B 0,C 180,E1 -19350,E2 -19350} C_VEL
LIN {X 0,Y 239.95,Z 309.809,A -85,B 0,C 180,E1 -19351.679,E2 -19351.679} C_VEL
LIN {X 0,Y 240.051,Z 309.223,A -85,B 0,C 180,E1 -19353.357,E2 -19353.357} C_VEL
LIN {X 0,Y 240.49,Z 306.9,A -85,B 0,C 180,E1 -19356.713,E2 -19356.713} C_VEL
LIN {X 0,Y 241.119,Z 304.034,A -85,B 0,C 180,E1 -19359.225,E2 -19359.225} C_VEL
LIN {X 0,Y 242.032,Z 300.146,A -85,B 0,C 180,E1 -19361.728,E2 -19361.728} C_VEL
LIN {X 0,Y 243.337,Z 295.127,A -85,B 0,C 180,E1 -19364.211,E2 -19364.211} C_VEL
LIN {X 0,Y 244.99,Z 288.804,A -85,B 0,C 180,E1 -19366.671,E2 -19366.671} C_VEL
LIN {X 0,Y 247.128,Z 280.887,A -85,B 0,C 180,E1 -19369.09,E2 -19369.09} C_VEL
LIN {X 0,Y 249.077,Z 272.922,A -85,B 0,C 180,E1 -19371.06,E2 -19371.06} C_VEL
LIN {X 0,Y 250.853,Z 264.043,A -85,B 0,C 180,E1 -19372.875,E2 -19372.875} C_VEL
LIN {X 0,Y 253.073,Z 253.277,A -85,B 0,C 180,E1 -19374.618,E2 -19374.618} C_VEL
LIN {X 0,Y 252.911,Z 248.944,A -85,B 0,C 180,E1 -19375.313,E2 -19375.313} C_VEL
LIN {X 0,Y 251.383,Z 238.215,A -85,B 0,C 180,E1 -19376.942,E2 -19376.942} C_VEL
LIN {X 0,Y 248.979,Z 227.371,A -85,B 0,C 180,E1 -19378.4,E2 -19378.4} C_VEL
LIN {X 0,Y 245.344,Z 215.366,A -85,B 0,C 180,E1 -19379.838,E2 -19379.838} C_VEL
LIN {X 0,Y 241.965,Z 206.056,A -85,B 0,C 180,E1 -19380.841,E2 -19380.841} C_VEL
LIN {X 0,Y 241.9,Z 205.693,A -85,B 0,C 180,E1 -19380.941,E2 -19380.941} C_VEL
LIN {X 0,Y 242.273,Z 202.094,A -85,B 0,C 180,E1 -19385.463,E2 -19385.463} C_VEL
LIN {X 0,Y 242.25,Z 199.892,A -85,B 0,C 180,E1 -19388.435,E2 -19388.435} C_VEL
LIN {X 0,Y 241.947,Z 197.491,A -85,B 0,C 180,E1 -19391.921,E2 -19391.921} C_VEL
LIN {X 0,Y 241.926,Z 197.349,A -85,B 0,C 180,E1 -19396.574,E2 -19396.574} C_VEL
LIN {X 0,Y 241.958,Z 197.346,A -85,B 0,C 180,E1 -19400.281,E2 -19400.281} C_VEL
LIN {X 0,Y 241.981,Z 197.344,A -85,B 0,C 180,E1 -19404.488,E2 -19404.488} C_VEL
LIN {X 0,Y 241.975,Z 197.343,A -85,B 0,C 180,E1 -19408.48,E2 -19408.48} C_VEL
LIN {X 0,Y 242.005,Z 197.342,A -85,B 0,C 180,E1 -19412.312,E2 -19412.312} C_VEL
LIN {X 0,Y 242.059,Z 197.334,A -85,B 0,C 180,E1 -19416.016,E2 -19416.016} C_VEL
LIN {X 0,Y 242.04,Z 197.335,A -85,B 0,C 180,E1 -19419.608,E2 -19419.608} C_VEL
LIN {X 0,Y 242.165,Z 197.317,A -85,B 0,C 180,E1 -19423.278,E2 -19423.278} C_VEL
LIN {X 0,Y 242.181,Z 197.317,A -85,B 0,C 180,E1 -19428.279,E2 -19428.279} C_VEL
LIN {X 0,Y 242.386,Z 197.294,A -85,B 0,C 180,E1 -19431.664,E2 -19431.664} C_VEL
LIN {X 0,Y 242.241,Z 197.311,A -85,B 0,C 180,E1 -19435.007,E2 -19435.007} C_VEL
LIN {X 0,Y 242.636,Z 197.259,A -85,B 0,C 180,E1 -19438.34,E2 -19438.34} C_VEL
LIN {X 0,Y 242.636,Z 197.261,A -85,B 0,C 180,E1 -19441.66,E2 -19441.66} C_VEL
LIN {X 0,Y 242.4,Z 197.293,A -85,B 0,C 180,E1 -19446.66,E2 -19446.66} C_VEL
LIN {X 0,Y 242.269,Z 197.306,A -85,B 0,C 180,E1 -19450.024,E2 -19450.024} C_VEL
LIN {X 0,Y 242.169,Z 197.321,A -85,B 0,C 180,E1 -19455.141,E2 -19455.141} C_VEL
LIN {X 0,Y 242.073,Z 197.333,A -85,B 0,C 180,E1 -19458.624,E2 -19458.624} C_VEL
LIN {X 0,Y 242.008,Z 197.34,A -85,B 0,C 180,E1 -19462.18,E2 -19462.18} C_VEL
LIN {X 0,Y 242.068,Z 197.333,A -85,B 0,C 180,E1 -19465.838,E2 -19465.838} C_VEL
LIN {X 0,Y 242.009,Z 197.342,A -85,B 0,C 180,E1 -19469.583,E2 -19469.583} C_VEL
LIN {X 0,Y 241.982,Z 197.346,A -85,B 0,C 180,E1 -19473.492,E2 -19473.492} C_VEL
LIN {X 0,Y 242.007,Z 197.364,A -85,B 0,C 180,E1 -19477.979,E2 -19477.979} C_VEL
LIN {X 0,Y 242.482,Z 200.45,A -85,B 0,C 180,E1 -19481.807,E2 -19481.807} C_VEL
LIN {X 0,Y 242.767,Z 202.004,A -85,B 0,C 180,E1 -19483.638,E2 -19483.638} C_VEL
LIN {X 0,Y 242.325,Z 203.311,A -85,B 0,C 180,E1 -19484.993,E2 -19484.993} C_VEL
LIN {X 0,Y 239.886,Z 205.782,A -85,B 0,C 180,E1 -19487.198,E2 -19487.198} C_VEL
LIN {X 0,Y 237.043,Z 208.818,A -85,B 0,C 180,E1 -19489.907,E2 -19489.907} C_VEL
LIN {X 0,Y 236.793,Z 209.756,A -85,B 0,C 180,E1 -19490.844,E2 -19490.844} C_VEL
LIN {X 0,Y 236.823,Z 212.456,A -85,B 0,C 180,E1 -19493.592,E2 -19493.592} C_VEL
LIN {X 0,Y 236.46,Z 215.256,A -85,B 0,C 180,E1 -19496.326,E2 -19496.326} C_VEL
LIN {X 0,Y 235.991,Z 217.332,A -85,B 0,C 180,E1 -19498.276,E2 -19498.276} C_VEL
LIN {X 0,Y 238.594,Z 226.532,A -85,B 0,C 180,E1 -19499.185,E2 -19499.185} C_VEL
LIN {X 0,Y 241.295,Z 237.807,A -85,B 0,C 180,E1 -19500.434,E2 -19500.434} C_VEL
LIN {X 0,Y 243.331,Z 249.868,A -85,B 0,C 180,E1 -19501.959,E2 -19501.959} C_VEL
LIN {X 0,Y 244.316,Z 260.796,A -85,B 0,C 180,E1 -19503.54,E2 -19503.54} C_VEL
LIN {X 0,Y 244.572,Z 271.701,A -85,B 0,C 180,E1 -19505.375,E2 -19505.375} C_VEL
LIN {X 0,Y 242.624,Z 280.62,A -85,B 0,C 180,E1 -19506.98,E2 -19506.98} C_VEL
LIN {X 0,Y 240.402,Z 289.782,A -85,B 0,C 180,E1 -19509.015,E2 -19509.015} C_VEL
LIN {X 0,Y 238.216,Z 298.718,A -85,B 0,C 180,E1 -19511.509,E2 -19511.509} C_VEL
LIN {X 0,Y 236.31,Z 305.908,A -85,B 0,C 180,E1 -19514.032,E2 -19514.032} C_VEL
LIN {X 0,Y 234.996,Z 310.762,A -85,B 0,C 180,E1 -19516.157,E2 -19516.157} C_VEL
LIN {X 0,Y 233.953,Z 315.488,A -85,B 0,C 180,E1 -19518.74,E2 -19518.74} C_VEL
LIN {X 0,Y 233.24,Z 319.101,A -85,B 0,C 180,E1 -19521.334,E2 -19521.334} C_VEL
LIN {X 0,Y 232.927,Z 320.964,A -85,B 0,C 180,E1 -19523.068,E2 -19523.068} C_VEL
LIN {X 0,Y 232.725,Z 322.656,A -85,B 0,C 180,E1 -19525.248,E2 -19525.248} C_VEL
LIN {X 0,Y 232.748,Z 323.976,A -85,B 0,C 180,E1 -19528.269,E2 -19528.269} C_VEL
LIN {X 0,Y 232.783,Z 324.192,A -85,B 0,C 180,E1 -19530,E2 -19530} C_VEL
LIN {X 0,Y 232.748,Z 323.969,A -85,B 0,C 180,E1 -19531.73,E2 -19531.73} C_VEL
LIN {X 0,Y 232.767,Z 322.348,A -85,B 0,C 180,E1 -19535.197,E2 -19535.197} C_VEL
LIN {X 0,Y 232.926,Z 320.941,A -85,B 0,C 180,E1 -19536.932,E2 -19536.932} C_VEL
LIN {X 0,Y 233.441,Z 317.991,A -85,B 0,C 180,E1 -19539.531,E2 -19539.531} C_VEL
LIN {X 0,Y 234.284,Z 314.003,A -85,B 0,C 180,E1 -19542.121,E2 -19542.121} C_VEL
LIN {X 0,Y 235.767,Z 307.875,A -85,B 0,C 180,E1 -19545.119,E2 -19545.119} C_VEL
LIN {X 0,Y 237.522,Z 301.188,A -85,B 0,C 180,E1 -19547.655,E2 -19547.655} C_VEL
LIN {X 0,Y 239.466,Z 293.837,A -85,B 0,C 180,E1 -19549.89,E2 -19549.89} C_VEL
LIN {X 0,Y 241.659,Z 284.389,A -85,B 0,C 180,E1 -19552.214,E2 -19552.214} C_VEL
LIN {X 0,Y 243.885,Z 275.066,A -85,B 0,C 180,E1 -19554.018,E2 -19554.018} C_VEL
LIN {X 0,Y 244.528,Z 271.529,A -85,B 0,C 180,E1 -19554.629,E2 -19554.629} C_VEL
LIN {X 0,Y 244.349,Z 261.895,A -85,B 0,C 180,E1 -19556.26,E2 -19556.26} C_VEL
LIN {X 0,Y 243.431,Z 250.802,A -85,B 0,C 180,E1 -19557.883,E2 -19557.883} C_VEL
LIN {X 0,Y 241.728,Z 239.867,A -85,B 0,C 180,E1 -19559.282,E2 -19559.282} C_VEL
LIN {X 0,Y 238.743,Z 227.031,A -85,B 0,C 180,E1 -19560.72,E2 -19560.72} C_VEL
LIN {X 0,Y 236.027,Z 218.04,A -85,B 0,C 180,E1 -19561.625,E2 -19561.625} C_VEL
LIN {X 0,Y 235.972,Z 217.294,A -85,B 0,C 180,E1 -19561.724,E2 -19561.724} C_VEL
LIN {X 0,Y 236.742,Z 213.456,A -85,B 0,C 180,E1 -19565.371,E2 -19565.371} C_VEL
LIN {X 0,Y 236.859,Z 210.298,A -85,B 0,C 180,E1 -19568.542,E2 -19568.542} C_VEL
LIN {X 0,Y 236.459,Z 207.062,A -85,B 0,C 180,E1 -19572.008,E2 -19572.008} C_VEL
LIN {X 0,Y 235.738,Z 202.972,A -85,B 0,C 180,E1 -19576.71,E2 -19576.71} C_VEL
LIN {X 0,Y 235.154,Z 199.44,A -85,B 0,C 180,E1 -19581.125,E2 -19581.125} C_VEL
LIN {X 0,Y 234.911,Z 198.225,A -85,B 0,C 180,E1 -19582.98,E2 -19582.98} C_VEL
LIN {X 0,Y 234.954,Z 198.219,A -85,B 0,C 180,E1 -19587.424,E2 -19587.424} C_VEL
LIN {X 0,Y 234.935,Z 198.22,A -85,B 0,C 180,E1 -19591.404,E2 -19591.404} C_VEL
LIN {X 0,Y 234.976,Z 198.217,A -85,B 0,C 180,E1 -19595.245,E2 -19595.245} C_VEL
LIN {X 0,Y 234.997,Z 198.214,A -85,B 0,C 180,E1 -19598.968,E2 -19598.968} C_VEL
LIN {X 0,Y 235.095,Z 198.202,A -85,B 0,C 180,E1 -19603.059,E2 -19603.059} C_VEL
LIN {X 0,Y 235.112,Z 198.196,A -85,B 0,C 180,E1 -19607.922,E2 -19607.922} C_VEL
LIN {X 0,Y 235.309,Z 198.175,A -85,B 0,C 180,E1 -19611.412,E2 -19611.412} C_VEL
LIN {X 0,Y 235.201,Z 198.189,A -85,B 0,C 180,E1 -19614.857,E2 -19614.857} C_VEL
LIN {X 0,Y 235.592,Z 198.137,A -85,B 0,C 180,E1 -19618.291,E2 -19618.291} C_VEL
LIN {X 0,Y 235.592,Z 198.137,A -85,B 0,C 180,E1 -19621.71,E2 -19621.71} C_VEL
LIN {X 0,Y 235.353,Z 198.167,A -85,B 0,C 180,E1 -19626.86,E2 -19626.86} C_VEL
LIN {X 0,Y 235.213,Z 198.185,A -85,B 0,C 180,E1 -19630.328,E2 -19630.328} C_VEL
LIN {X 0,Y 235.112,Z 198.197,A -85,B 0,C 180,E1 -19635.607,E2 -19635.607} C_VEL
LIN {X 0,Y 235.008,Z 198.21,A -85,B 0,C 180,E1 -19639.206,E2 -19639.206} C_VEL
LIN {X 0,Y 234.96,Z 198.216,A -85,B 0,C 180,E1 -19642.883,E2 -19642.883} C_VEL
LIN {X 0,Y 234.968,Z 198.216,A -85,B 0,C 180,E1 -19646.658,E2 -19646.658} C_VEL
LIN {X 0,Y 234.93,Z 198.22,A -85,B 0,C 180,E1 -19650.568,E2 -19650.568} C_VEL
LIN {X 0,Y 234.925,Z 198.222,A -85,B 0,C 180,E1 -19654.639,E2 -19654.639} C_VEL
LIN {X 0,Y 234.941,Z 198.224,A -85,B 0,C 180,E1 -19658.945,E2 -19658.945} C_VEL
LIN {X 0,Y 234.878,Z 198.229,A -85,B 0,C 180,E1 -19663.489,E2 -19663.489} C_VEL
LIN {X 0,Y 234.878,Z 198.229,A -85,B 0,C 180,E1 -19666.513,E2 -19666.513} C_VEL
LIN {X 0,Y 235.033,Z 199.142,A -85,B 0,C 180,E1 -19668.865,E2 -19668.865} C_VEL
LIN {X 0,Y 235.224,Z 200.668,A -85,B 0,C 180,E1 -19671.14,E2 -19671.14} C_VEL
LIN {X 0,Y 235.261,Z 202.548,A -85,B 0,C 180,E1 -19673.763,E2 -19673.763} C_VEL
LIN {X 0,Y 234.987,Z 206.05,A -85,B 0,C 180,E1 -19678.269,E2 -19678.269} C_VEL
LIN {X 0,Y 236.038,Z 209.212,A -85,B 0,C 180,E1 -19678.595,E2 -19678.595} C_VEL
LIN {X 0,Y 240.358,Z 221.248,A -85,B 0,C 180,E1 -19680.046,E2 -19680.046} C_VEL
LIN {X 0,Y 243.544,Z 233.153,A -85,B 0,C 180,E1 -19681.623,E2 -19681.623} C_VEL
LIN {X 0,Y 245.426,Z 243.229,A -85,B 0,C 180,E1 -19683.114,E2 -19683.114} C_VEL
LIN {X 0,Y 246.494,Z 252.702,A -85,B 0,C 180,E1 -19684.68,E2 -19684.68} C_VEL
LIN {X 0,Y 245.433,Z 259.068,A -85,B 0,C 180,E1 -19685.693,E2 -19685.693} C_VEL
LIN {X 0,Y 243.247,Z 268.968,A -85,B 0,C 180,E1 -19687.537,E2 -19687.537} C_VEL
LIN {X 0,Y 241.275,Z 277.595,A -85,B 0,C 180,E1 -19689.541,E2 -19689.541} C_VEL
LIN {X 0,Y 238.953,Z 286.207,A -85,B 0,C 180,E1 -19692.012,E2 -19692.012} C_VEL
LIN {X 0,Y 237.107,Z 293.068,A -85,B 0,C 180,E1 -19694.529,E2 -19694.529} C_VEL
LIN {X 0,Y 235.546,Z 298.562,A -85,B 0,C 180,E1 -19697.069,E2 -19697.069} C_VEL
LIN {X 0,Y 234.392,Z 302.871,A -85,B 0,C 180,E1 -19699.636,E2 -19699.636} C_VEL
LIN {X 0,Y 233.856,Z 305.148,A -85,B 0,C 180,E1 -19701.358,E2 -19701.358} C_VEL
LIN {X 0,Y 233.315,Z 307.56,A -85,B 0,C 180,E1 -19703.743,E2 -19703.743} C_VEL
LIN {X 0,Y 232.979,Z 309.379,A -85,B 0,C 180,E1 -19706.542,E2 -19706.542} C_VEL
LIN {X 0,Y 232.838,Z 310.215,A -85,B 0,C 180,E1 -19710,E2 -19710} C_VEL
LIN {X 0,Y 232.864,Z 310.022,A -85,B 0,C 180,E1 -19711.73,E2 -19711.73} C_VEL
LIN {X 0,Y 232.977,Z 309.435,A -85,B 0,C 180,E1 -19713.459,E2 -19713.459} C_VEL
LIN {X 0,Y 233.433,Z 307.113,A -85,B 0,C 180,E1 -19716.917,E2 -19716.917} C_VEL
LIN {X 0,Y 234.096,Z 304.246,A -85,B 0,C 180,E1 -19719.505,E2 -19719.505} C_VEL
LIN {X 0,Y 235.074,Z 300.358,A -85,B 0,C 180,E1 -19722.08,E2 -19722.08} C_VEL
LIN {X 0,Y 236.459,Z 295.338,A -85,B 0,C 180,E1 -19724.634,E2 -19724.634} C_VEL
LIN {X 0,Y 238.202,Z 289.015,A -85,B 0,C 180,E1 -19727.161,E2 -19727.161} C_VEL
LIN {X 0,Y 240.439,Z 281.097,A -85,B 0,C 180,E1 -19729.642,E2 -19729.642} C_VEL
LIN {X 0,Y 242.548,Z 272.587,A -85,B 0,C 180,E1 -19731.793,E2 -19731.793} C_VEL
LIN {X 0,Y 244.604,Z 263.184,A -85,B 0,C 180,E1 -19733.719,E2 -19733.719} C_VEL
LIN {X 0,Y 246.632,Z 253.486,A -85,B 0,C 180,E1 -19735.305,E2 -19735.305} C_VEL
LIN {X 0,Y 245.331,Z 242.529,A -85,B 0,C 180,E1 -19737.123,E2 -19737.123} C_VEL
LIN {X 0,Y 243.452,Z 232.593,A -85,B 0,C 180,E1 -19738.584,E2 -19738.584} C_VEL
LIN {X 0,Y 240.236,Z 220.935,A -85,B 0,C 180,E1 -19740.134,E2 -19740.134} C_VEL
LIN {X 0,Y 236.087,Z 209.282,A -85,B 0,C 180,E1 -19741.534,E2 -19741.534} C_VEL
LIN {X 0,Y 234.968,Z 205.946,A -85,B 0,C 180,E1 -19741.933,E2 -19741.933} C_VEL
LIN {X 0,Y 235.267,Z 202.658,A -85,B 0,C 180,E1 -19746.239,E2 -19746.239} C_VEL
LIN {X 0,Y 235.192,Z 200.677,A -85,B 0,C 180,E1 -19749.019,E2 -19749.019} C_VEL
LIN {X 0,Y 234.979,Z 198.951,A -85,B 0,C 180,E1 -19751.606,E2 -19751.606} C_VEL
LIN {X 0,Y 234.876,Z 198.226,A -85,B 0,C 180,E1 -19754.099,E2 -19754.099} C_VEL
LIN {X 0,Y 234.883,Z 198.228,A -85,B 0,C 180,E1 -19758.832,E2 -19758.832} C_VEL
LIN {X 0,Y 234.919,Z 198.223,A -85,B 0,C 180,E1 -19761.079,E2 -19761.079} C_VEL
LIN {X 0,Y 234.927,Z 198.221,A -85,B 0,C 180,E1 -19765.361,E2 -19765.361} C_VEL
LIN {X 0,Y 234.924,Z 198.221,A -85,B 0,C 180,E1 -19769.431,E2 -19769.431} C_VEL
